RoboDK station: DensoAssembly.rdk

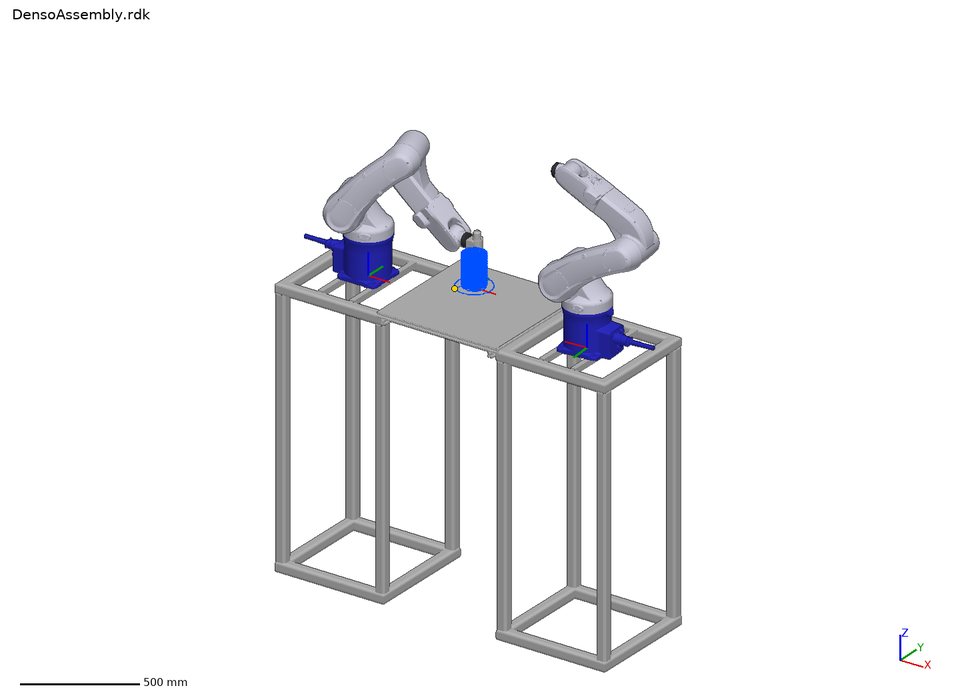
[picture v0: the station drawn from its stored meshes, robots at their saved joint values, targets as dots, program paths as lines]
Station DensoAssembly (saved by RoboDK 5.5.4). Poses are relative to the parent item; angles as X-Y-Z fixed-axis rotations.
Station parameters (name, value as stored): TAGS, ['Additive Manufacturing', 'Additive manufacturing']
  - frame Denso VS-6577G-B Base at (0, -10, -20) mm
    - robot Denso VS-6577G-B: 6 axes, payload 7 kg, reach 854 mm, repeatability 0.03 mm, weight 36 kg
        modified DH rows (alpha deg, a mm, theta deg, d mm): 0, 0, 0, 335; -90, 75, -90, 0; 0, 365, -90, 0; -90, 90, 0, 405; 90, 0, 0, 0; -90, 0, 0, 80
        joint limits [-170, -100, -119, -190, -120, -360] to [170, 135, 169, 190, 120, 360]; home [0, 0, 90, 0, 0, 0]; saved at [-161.491, -43.825, -94.782, 24.049, 51.169, -15.633]
      - tool NCRDK, TCP at (55, 0, 30) mm, rotated rx 0 ry 90 rz 0 deg, size 57.1 x 107.2 x 69.8 mm, geometry from NCRDK.STL
    - object Table 1400x800x800mm at (-100, 160, 0) mm, size 1420 x 820 x 800 mm, geometry from Table-1400x800x800mm.sld
    - object RobotStand_SWP at (50, -240, -710) mm, size 609.6 x 1373.2 x 1689.1 mm, geometry from RobotStand_SWP.STEP
  - frame Reference at (454.66, 114.92, 0) mm
    - object Part at (0, 0, 0) mm, size 120 x 120 x 160 mm, geometry from part.sld
  - machining project Print3D settings: C:/Users/Albert/AppData/Local/Temp/Part.stl | rotZ(0) | rotX(0)*rotY(0) | rotZ(0)
  - program Print3D (7572 instructions, listed below)
  - Python program Extruder (listed below)
  - Python program SimulateFinalResult (listed below)
  - frame Denso VS-6577G-B Base at (1145.1, -47.51, -20) mm, rotated rx 0 ry 0 rz -175.68 deg
    - robot Denso VS-6577G-B: 6 axes, payload 7 kg, reach 854 mm, repeatability 0.03 mm, weight 36 kg
        modified DH rows (alpha deg, a mm, theta deg, d mm): 0, 0, 0, 335; -90, 75, -90, 0; 0, 365, -90, 0; -90, 90, 0, 405; 90, 0, 0, 0; -90, 0, 0, 80
        joint limits [-170, -100, -119, -190, -120, -360] to [170, 135, 169, 190, 120, 360]; home [0, 0, 90, 0, 0, 0]; saved at [0, -58.32, 121.453, 0, 26.867, 0]
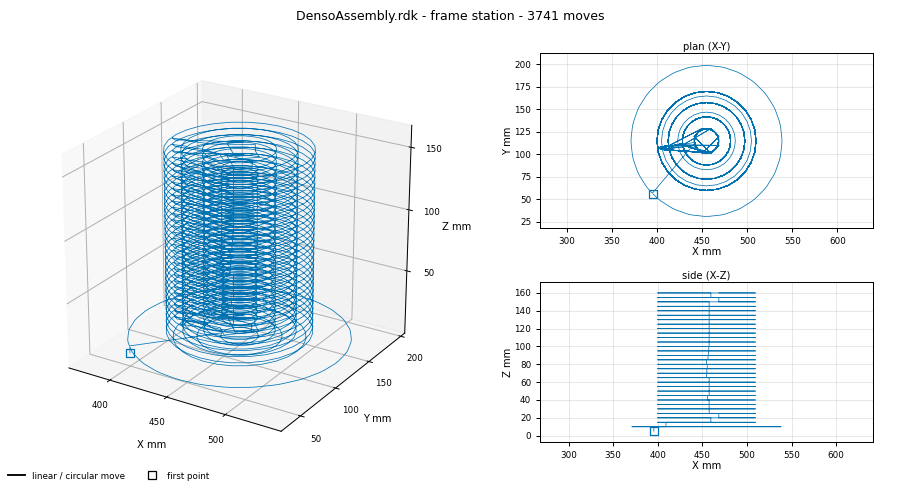
[picture p0: tool path of DensoAssembly.rdk in frame station, 3741 of 3741 moves have a stored position in this frame; points joined in program order, loops and branches not executed]

--- program Print3D (robot Denso VS-6577G-B) ---
  Set speed (83.3 mm/s)
  Set speed (1000.0 mm/s)
  Set Ref.: Reference
  Set Tool: NCRDK
  Show NCRDK
  MoveJ 1 to (-59.03, -59.03, 5) mm, rotated rx 180 ry 0 rz 180 deg; joints [-167.009, -64.344, -97.717, 13.631, 72.535, -4.163]
  MoveL 2 to (-59.03, -59.03, 5) mm, rotated rx 180 ry 0 rz 180 deg; joints [-167.009, -64.344, -97.717, 13.631, 72.535, -4.163]
  Call Extruder(-1)
  MoveL 3 to (-59.03, -59.03, 5) mm, rotated rx 180 ry 0 rz 180 deg; joints [-167.009, -64.344, -97.717, 13.631, 72.535, -4.163]
  Call Extruder(0.00000)
  Set speed (130.0 mm/s)
  MoveL 4 to (-59.03, -59.03, 10) mm, rotated rx 180 ry 0 rz 180 deg; joints [-167.009, -63.51, -98.227, 13.655, 72.22, -4.243]
  Call Extruder(-2.00000)
  Set speed (40.0 mm/s)
  MoveL 5 to (-59.03, -59.03, 10) mm, rotated rx 180 ry 0 rz 180 deg; joints [-167.009, -63.51, -98.227, 13.655, 72.22, -4.243]
  Call Extruder(0.00000)
  Set speed (130.0 mm/s)
  MoveL 6 to (-59.03, -59.03, 10) mm, rotated rx 180 ry 0 rz 180 deg; joints [-167.009, -63.51, -98.227, 13.655, 72.22, -4.243]
  Call Extruder(2.00000)
  Set speed (40.0 mm/s)
  MoveL 7 to (-59.03, -59.03, 10) mm, rotated rx 180 ry 0 rz 180 deg; joints [-167.009, -63.51, -98.227, 13.655, 72.22, -4.243]
  Call Extruder(25.86117)
  Set speed (30.0 mm/s)
  MoveL 8 to (-54.28, -63.78, 10) mm, rotated rx 180 ry 0 rz 180 deg; joints [-168.109, -63.573, -97.687, 12.537, 71.677, -3.999]
  Call Extruder(44.83322)
  MoveL 9 to (-50.1, -67.11, 10) mm, rotated rx 180 ry 0 rz 180 deg; joints [-168.895, -63.638, -97.171, 11.741, 71.182, -3.835]
  Call Extruder(92.55677)
  MoveL 10 to (-38.72, -74.26, 10) mm, rotated rx 180 ry 0 rz 176 deg; joints [-169.213, -63.884, -95.415, 15.759, 70.015, -5.509]
  Call Extruder(111.53101)
  MoveL 11 to (-33.91, -76.57, 10) mm, rotated rx 180 ry 0 rz 176 deg; joints [-169.789, -63.989, -94.75, 15.203, 69.419, -5.457]
  Call Extruder(159.25391)
  MoveL 12 to (-21.23, -81.01, 10) mm, rotated rx 180 ry 0 rz 172 deg; joints [-169.657, -64.367, -92.58, 19.815, 68.18, -7.628]
  Call Extruder(178.22553)
  MoveL 13 to (-16.02, -82.2, 10) mm, rotated rx 180 ry 0 rz 168 deg; joints [-168.792, -64.603, -91.363, 25.148, 68.018, -9.967]
  Call Extruder(225.94862)
  MoveL 14 to (-2.67, -83.7, 10) mm, rotated rx -180 ry 0 rz 168 deg; joints [-169.458, -65.044, -89.278, 24.729, 66.409, -10.444]
  Call Extruder(244.92246)
  MoveL 15 to (2.67, -83.7, 10) mm, rotated rx 180 ry 0 rz 168 deg; joints [-169.615, -65.24, -88.41, 24.684, 65.77, -10.682]
  Call Extruder(246.41380)
  MoveL 16 to (3.09, -83.66, 10) mm, rotated rx 180 ry 0 rz 168 deg; joints [-169.62, -65.256, -88.341, 24.689, 65.72, -10.704]
  Call Extruder(292.64546)
  MoveL 17 to (16.02, -82.2, 10) mm, rotated rx 180 ry 0 rz 168 deg; joints [-169.759, -65.781, -86.16, 24.862, 64.19, -11.406]
  Call Extruder(311.61718)
  MoveL 18 to (21.23, -81.01, 10) mm, rotated rx 180 ry 0 rz 168 deg; joints [-169.722, -66.013, -85.248, 25.044, 63.581, -11.744]
  Call Extruder(359.33987)
  MoveL 19 to (33.91, -76.57, 10) mm, rotated rx -180 ry 0 rz 168 deg; joints [-169.411, -66.628, -82.943, 25.757, 62.12, -12.714]
  Call Extruder(378.31438)
  MoveL 20 to (38.72, -74.26, 10) mm, rotated rx -180 ry 0 rz 168 deg; joints [-169.208, -66.882, -82.031, 26.136, 61.575, -13.147]
  Call Extruder(426.03771)
  MoveL 21 to (50.1, -67.11, 10) mm, rotated rx -180 ry 0 rz 172 deg; joints [-169.533, -67.389, -80.276, 21.566, 59.513, -11.339]
  Call Extruder(445.00995)
  MoveL 22 to (54.28, -63.78, 10) mm, rotated rx 180 ry 0 rz 172 deg; joints [-169.179, -67.643, -79.418, 22.103, 59.025, -11.806]
  Call Extruder(492.73236)
  MoveL 23 to (63.78, -54.28, 10) mm, rotated rx 180 ry 0 rz 176 deg; joints [-169.152, -68.143, -77.78, 17.748, 57.208, -9.834]
  Call Extruder(511.70474)
  MoveL 24 to (67.11, -50.1, 10) mm, rotated rx -180 ry 0 rz -180 deg; joints [-169.701, -68.281, -77.339, 12.417, 56.249, -6.974]
  Call Extruder(559.42802)
  MoveL 25 to (74.26, -38.72, 10) mm, rotated rx 180 ry 0 rz 180 deg; joints [-168.372, -68.831, -75.608, 14.195, 55.276, -8.199]
  Call Extruder(578.40244)
  MoveL 26 to (76.57, -33.91, 10) mm, rotated rx 180 ry 0 rz 180 deg; joints [-167.808, -69.033, -74.985, 14.95, 54.951, -8.718]
  Call Extruder(626.12508)
  MoveL 27 to (81.01, -21.23, 10) mm, rotated rx 180 ry 0 rz 180 deg; joints [-166.309, -69.49, -73.602, 16.944, 54.305, -10.08]
  Call Extruder(645.09694)
  MoveL 28 to (82.2, -16.02, 10) mm, rotated rx 180 ry 0 rz -180 deg; joints [-165.688, -69.648, -73.131, 17.765, 54.118, -10.635]
  Call Extruder(692.81987)
  MoveL 29 to (83.7, -2.67, 10) mm, rotated rx -180 ry 0 rz -180 deg; joints [-164.071, -69.976, -72.16, 19.875, 53.828, -12.044]
  Call Extruder(711.79372)
  MoveL 30 to (83.7, 2.67, 10) mm, rotated rx 180 ry 0 rz 180 deg; joints [-163.413, -70.078, -71.864, 20.722, 53.786, -12.599]
  Call Extruder(759.51663)
  MoveL 31 to (82.2, 16.02, 10) mm, rotated rx 180 ry 0 rz 180 deg; joints [-161.727, -70.253, -71.354, 22.845, 53.862, -13.953]
  Call Extruder(778.48846)
  MoveL 32 to (81.01, 21.23, 10) mm, rotated rx -180 ry 0 rz -180 deg; joints [-161.05, -70.29, -71.247, 23.678, 53.964, -14.465]
  Call Extruder(826.21114)
  MoveL 33 to (76.57, 33.91, 10) mm, rotated rx 180 ry 0 rz 180 deg; joints [-159.34, -70.299, -71.222, 25.719, 54.394, -15.666]
  Call Extruder(845.18561)
  MoveL 34 to (74.26, 38.72, 10) mm, rotated rx -180 ry 0 rz 180 deg; joints [-158.662, -70.268, -71.31, 26.502, 54.631, -16.099]
  Call Extruder(892.90887)
  MoveL 35 to (67.11, 50.1, 10) mm, rotated rx 180 ry 0 rz 180 deg; joints [-156.971, -70.109, -71.773, 28.382, 55.383, -17.063]
  Call Extruder(911.88119)
  MoveL 36 to (63.78, 54.28, 10) mm, rotated rx 180 ry 0 rz 180 deg; joints [-156.31, -70.014, -72.051, 29.087, 55.739, -17.389]
  Call Extruder(959.60361)
  MoveL 37 to (54.28, 63.78, 10) mm, rotated rx 180 ry 0 rz 180 deg; joints [-154.685, -69.699, -72.978, 30.745, 56.764, -18.056]
  Call Extruder(978.57593)
  MoveL 38 to (50.1, 67.11, 10) mm, rotated rx 180 ry 0 rz -180 deg; joints [-154.059, -69.547, -73.432, 31.353, 57.218, -18.257]
  Call Extruder(1026.29918)
  MoveL 39 to (38.72, 74.26, 10) mm, rotated rx -180 ry 0 rz 180 deg; joints [-152.546, -69.101, -74.778, 32.748, 58.459, -18.595]
  Call Extruder(1045.27367)
  MoveL 40 to (33.91, 76.57, 10) mm, rotated rx -180 ry 0 rz 180 deg; joints [-151.975, -68.903, -75.386, 33.246, 58.986, -18.663]
  Call Extruder(1092.99635)
  MoveL 41 to (21.23, 81.01, 10) mm, rotated rx -180 ry 0 rz -180 deg; joints [-150.627, -68.36, -77.086, 34.348, 60.378, -18.664]
  Call Extruder(1111.96805)
  MoveL 42 to (16.02, 82.2, 10) mm, rotated rx 180 ry 0 rz 180 deg; joints [-150.133, -68.131, -77.821, 34.725, 60.953, -18.599]
  Call Extruder(1159.69109)
  MoveL 43 to (2.67, 83.7, 10) mm, rotated rx 180 ry 0 rz -180 deg; joints [-149.008, -67.53, -79.796, 35.511, 62.434, -18.275]
  Call Extruder(1178.66494)
  MoveL 44 to (-2.67, 83.7, 10) mm, rotated rx 180 ry 0 rz 180 deg; joints [-148.615, -67.286, -80.624, 35.756, 63.03, -18.085]
  Call Extruder(1226.38787)
  MoveL 45 to (-16.02, 82.2, 10) mm, rotated rx 180 ry 0 rz -180 deg; joints [-147.779, -66.671, -82.786, 36.196, 64.538, -17.464]
  Call Extruder(1245.35974)
  MoveL 46 to (-21.23, 81.01, 10) mm, rotated rx -180 ry 0 rz -180 deg; joints [-147.514, -66.43, -83.669, 36.297, 65.134, -17.164]
  Call Extruder(1293.08238)
  MoveL 47 to (-33.91, 76.57, 10) mm, rotated rx 180 ry 0 rz 180 deg; joints [-147.039, -65.841, -85.922, 36.354, 66.611, -16.287]
  Call Extruder(1312.05679)
  MoveL 48 to (-38.72, 74.26, 10) mm, rotated rx -180 ry 0 rz 180 deg; joints [-146.933, -65.618, -86.82, 36.294, 67.184, -15.896]
  Call Extruder(1359.78007)
  MoveL 49 to (-50.1, 67.11, 10) mm, rotated rx -180 ry 0 rz 180 deg; joints [-146.898, -65.092, -89.06, 35.92, 68.579, -14.819]
  Call Extruder(1378.75242)
  MoveL 50 to (-54.28, 63.78, 10) mm, rotated rx 180 ry 0 rz -180 deg; joints [-146.982, -64.901, -89.932, 35.678, 69.11, -14.361]
  Call Extruder(1380.24377)
  MoveL 51 to (-54.57, 63.48, 10) mm, rotated rx 180 ry 0 rz 180 deg; joints [-146.997, -64.886, -89.999, 35.652, 69.149, -14.322]
  Call Extruder(1426.47485)
  MoveL 52 to (-63.78, 54.28, 10) mm, rotated rx 180 ry 0 rz -180 deg; joints [-147.462, -64.468, -92.052, 34.822, 70.373, -13.151]
  Call Extruder(1445.44710)
  MoveL 53 to (-67.11, 50.1, 10) mm, rotated rx 180 ry 0 rz -180 deg; joints [-147.764, -64.316, -92.854, 34.38, 70.841, -12.656]
  Call Extruder(1493.17037)
  MoveL 54 to (-74.26, 38.72, 10) mm, rotated rx 180 ry 0 rz 180 deg; joints [-148.817, -63.99, -94.742, 33.001, 71.922, -11.394]
  Call Extruder(1512.14494)
  MoveL 55 to (-76.57, 33.91, 10) mm, rotated rx 180 ry 0 rz 180 deg; joints [-149.354, -63.882, -95.431, 32.347, 72.307, -10.895]
  Call Extruder(1559.86760)
  MoveL 56 to (-81.01, 21.23, 10) mm, rotated rx -180 ry 0 rz -180 deg; joints [-150.998, -63.662, -96.979, 30.438, 73.148, -9.667]
  Call Extruder(1578.83925)
  MoveL 57 to (-82.2, 16.02, 10) mm, rotated rx 180 ry 0 rz -180 deg; joints [-151.763, -63.595, -97.512, 29.58, 73.425, -9.198]
  Call Extruder(1626.56228)
  MoveL 58 to (-83.7, 2.67, 10) mm, rotated rx -180 ry 0 rz 180 deg; joints [-153.943, -63.467, -98.621, 27.197, 73.961, -8.081]
  Call Extruder(1645.53608)
  MoveL 59 to (-83.7, -2.67, 10) mm, rotated rx -180 ry 0 rz -180 deg; joints [-154.897, -63.432, -98.963, 26.175, 74.104, -7.667]
  Call Extruder(1693.25913)
  MoveL 60 to (-82.2, -16.02, 10) mm, rotated rx -180 ry 0 rz 180 deg; joints [-157.465, -63.375, -99.554, 23.464, 74.267, -6.713]
  Call Extruder(1712.23091)
  MoveL 61 to (-81.01, -21.23, 10) mm, rotated rx -180 ry 0 rz 180 deg; joints [-158.53, -63.363, -99.678, 22.352, 74.25, -6.368]
  Call Extruder(1759.95353)
  MoveL 62 to (-76.57, -33.91, 10) mm, rotated rx 180 ry 0 rz 180 deg; joints [-161.248, -63.361, -99.707, 19.539, 73.991, -5.59]
  Call Extruder(1778.92790)
  MoveL 63 to (-74.26, -38.72, 10) mm, rotated rx 180 ry 0 rz 180 deg; joints [-162.318, -63.37, -99.605, 18.438, 73.802, -5.314]
  Call Extruder(1826.65135)
  MoveL 64 to (-67.11, -50.1, 10) mm, rotated rx 180 ry 0 rz 180 deg; joints [-164.913, -63.421, -99.068, 15.785, 73.111, -4.695]
  Call Extruder(1845.62336)
  MoveL 65 to (-63.78, -54.28, 10) mm, rotated rx 180 ry 0 rz -180 deg; joints [-165.882, -63.454, -98.747, 14.798, 72.756, -4.478]
  Call Extruder(1864.15697)
  MoveL 66 to (-60.09, -57.97, 10) mm, rotated rx -180 ry 0 rz 180 deg; joints [-166.759, -63.497, -98.345, 13.908, 72.341, -4.296]
  Call Extruder(1862.15697)
  Set speed (40.0 mm/s)
  MoveL 67 to (-60.09, -57.97, 10) mm, rotated rx -180 ry 0 rz 180 deg; joints [-166.759, -63.497, -98.345, 13.908, 72.341, -4.296]
  Call Extruder(0.00000)
  Set speed (130.0 mm/s)
  MoveL 68 to (-13.65, -3.12, 10) mm, rotated rx -180 ry 0 rz 180 deg; joints [-159.797, -65.133, -88.882, 22.263, 65.721, -9.555]
  Call Extruder(2.00000)
  Set speed (40.0 mm/s)
  MoveL 69 to (-13.65, -3.12, 10) mm, rotated rx -180 ry 0 rz 180 deg; joints [-159.797, -65.133, -88.882, 22.263, 65.721, -9.555]
  Call Extruder(13.13706)
  Set speed (30.0 mm/s)
  MoveL 70 to (-12.62, -6.08, 10) mm, rotated rx 180 ry 0 rz 180 deg; joints [-160.306, -65.131, -88.888, 21.711, 65.641, -9.326]
  Call Extruder(24.27428)
  MoveL 71 to (-10.95, -8.73, 10) mm, rotated rx -180 ry 0 rz 180 deg; joints [-160.802, -65.157, -88.774, 21.188, 65.48, -9.139]
  Call Extruder(35.41276)
  MoveL 72 to (-8.73, -10.95, 10) mm, rotated rx -180 ry 0 rz 180 deg; joints [-161.258, -65.209, -88.546, 20.721, 65.244, -9.002]
  Call Extruder(46.54998)
  MoveL 73 to (-6.08, -12.62, 10) mm, rotated rx 180 ry 0 rz -180 deg; joints [-161.649, -65.285, -88.217, 20.337, 64.945, -8.92]
  Call Extruder(57.68705)
  MoveL 74 to (-3.12, -13.65, 10) mm, rotated rx -180 ry 0 rz 180 deg; joints [-161.955, -65.382, -87.802, 20.055, 64.6, -8.899]
  Call Extruder(68.82500)
  MoveL 75 to (0, -14, 10) mm, rotated rx -180 ry 0 rz 180 deg; joints [-162.16, -65.496, -87.324, 19.889, 64.225, -8.94]
  Call Extruder(79.96296)
  MoveL 76 to (3.12, -13.65, 10) mm, rotated rx -180 ry 0 rz 180 deg; joints [-162.258, -65.621, -86.806, 19.847, 63.842, -9.042]
  Call Extruder(91.10003)
  MoveL 77 to (6.08, -12.62, 10) mm, rotated rx 180 ry 0 rz 180 deg; joints [-162.244, -65.752, -86.276, 19.929, 63.468, -9.2]
  Call Extruder(102.23724)
  MoveL 78 to (8.73, -10.95, 10) mm, rotated rx 180 ry 0 rz -180 deg; joints [-162.124, -65.882, -85.759, 20.128, 63.124, -9.408]
  Call Extruder(113.37572)
  MoveL 79 to (10.95, -8.73, 10) mm, rotated rx 180 ry 0 rz 180 deg; joints [-161.905, -66.004, -85.281, 20.434, 62.826, -9.656]
  Call Extruder(124.51294)
  MoveL 80 to (12.62, -6.08, 10) mm, rotated rx -180 ry 0 rz 180 deg; joints [-161.6, -66.112, -84.866, 20.828, 62.59, -9.933]
  Call Extruder(135.65003)
  MoveL 81 to (13.65, -3.12, 10) mm, rotated rx 180 ry 0 rz 180 deg; joints [-161.224, -66.199, -84.533, 21.291, 62.427, -10.225]
  Call Extruder(146.78796)
  MoveL 82 to (14, 0, 10) mm, rotated rx 180 ry 0 rz 180 deg; joints [-160.796, -66.261, -84.3, 21.799, 62.345, -10.516]
  Call Extruder(157.92590)
  MoveL 83 to (13.65, 3.12, 10) mm, rotated rx 180 ry 0 rz 180 deg; joints [-160.336, -66.293, -84.178, 22.328, 62.347, -10.792]
  Call Extruder(169.06301)
  MoveL 84 to (12.62, 6.08, 10) mm, rotated rx 180 ry 0 rz 180 deg; joints [-159.864, -66.295, -84.172, 22.852, 62.432, -11.036]
  Call Extruder(180.20021)
  MoveL 85 to (10.95, 8.73, 10) mm, rotated rx 180 ry 0 rz 180 deg; joints [-159.401, -66.265, -84.283, 23.346, 62.597, -11.236]
  Call Extruder(191.33869)
  MoveL 86 to (8.73, 10.95, 10) mm, rotated rx -180 ry 0 rz -180 deg; joints [-158.969, -66.206, -84.506, 23.79, 62.831, -11.381]
  Call Extruder(202.47589)
  MoveL 87 to (6.08, 12.62, 10) mm, rotated rx 180 ry 0 rz -180 deg; joints [-158.587, -66.122, -84.829, 24.16, 63.124, -11.463]
  Call Extruder(213.61299)
  MoveL 88 to (3.12, 13.65, 10) mm, rotated rx 180 ry 0 rz 180 deg; joints [-158.274, -66.016, -85.237, 24.441, 63.462, -11.478]
  Call Extruder(224.75094)
  MoveL 89 to (0, 14, 10) mm, rotated rx 180 ry 0 rz -180 deg; joints [-158.046, -65.895, -85.709, 24.618, 63.827, -11.426]
  Call Extruder(235.88887)
  MoveL 90 to (-3.12, 13.65, 10) mm, rotated rx 180 ry 0 rz 180 deg; joints [-157.916, -65.765, -86.224, 24.682, 64.203, -11.31]
  Call Extruder(247.02595)
  MoveL 91 to (-6.08, 12.62, 10) mm, rotated rx 180 ry 0 rz -180 deg; joints [-157.892, -65.634, -86.754, 24.629, 64.57, -11.137]
  Call Extruder(258.16319)
  MoveL 92 to (-8.73, 10.95, 10) mm, rotated rx -180 ry 0 rz 180 deg; joints [-157.978, -65.508, -87.274, 24.458, 64.912, -10.916]
  Call Extruder(269.30166)
  MoveL 93 to (-10.95, 8.73, 10) mm, rotated rx -180 ry 0 rz 180 deg; joints [-158.173, -65.392, -87.757, 24.176, 65.211, -10.66]
  Call Extruder(280.43886)
  MoveL 94 to (-12.62, 6.08, 10) mm, rotated rx 180 ry 0 rz 180 deg; joints [-158.469, -65.294, -88.179, 23.795, 65.452, -10.381]
  Call Extruder(291.57594)
  MoveL 95 to (-13.65, 3.12, 10) mm, rotated rx 180 ry 0 rz 180 deg; joints [-158.852, -65.215, -88.518, 23.334, 65.623, -10.095]
  Call Extruder(302.71390)
  MoveL 96 to (-14, 0, 10) mm, rotated rx 180 ry 0 rz 180 deg; joints [-159.303, -65.161, -88.756, 22.814, 65.714, -9.816]
  Call Extruder(308.52395)
  MoveL 97 to (-13.82, -1.63, 10) mm, rotated rx 180 ry 0 rz 180 deg; joints [-159.56, -65.146, -88.822, 22.527, 65.718, -9.68]
  Set speed (130.0 mm/s)
  MoveL 98 to (-31.39, -5.11, 10) mm, rotated rx -180 ry 0 rz 180 deg; joints [-159.07, -64.537, -91.697, 22.68, 67.888, -8.939]
  Call Extruder(315.66877)
  Set speed (30.0 mm/s)
  MoveL 99 to (-31.17, -7.11, 10) mm, rotated rx -180 ry 0 rz 180 deg; joints [-159.404, -64.521, -91.777, 22.314, 67.896, -8.779]
  Call Extruder(341.09651)
  MoveL 100 to (-28.8, -13.87, 10) mm, rotated rx 180 ry 0 rz 180 deg; joints [-160.628, -64.518, -91.791, 21.005, 67.725, -8.281]
  Call Extruder(366.52461)
  MoveL 101 to (-24.99, -19.93, 10) mm, rotated rx 180 ry 0 rz 180 deg; joints [-161.818, -64.571, -91.526, 19.761, 67.358, -7.874]
  Call Extruder(391.95312)
  MoveL 102 to (-19.93, -25, 10) mm, rotated rx -180 ry 0 rz -180 deg; joints [-162.895, -64.677, -90.996, 18.661, 66.814, -7.574]
  Call Extruder(417.38123)
  MoveL 103 to (-13.87, -28.8, 10) mm, rotated rx 180 ry 0 rz -180 deg; joints [-163.797, -64.837, -90.232, 17.768, 66.122, -7.391]
  Call Extruder(442.80898)
  MoveL 104 to (-7.11, -31.17, 10) mm, rotated rx -180 ry 0 rz -180 deg; joints [-164.477, -65.045, -89.275, 17.13, 65.32, -7.333]
  Call Extruder(468.23739)
  MoveL 105 to (0, -31.97, 10) mm, rotated rx 180 ry 0 rz 180 deg; joints [-164.906, -65.295, -88.175, 16.775, 64.452, -7.407]
  Call Extruder(493.66579)
  MoveL 106 to (7.11, -31.17, 10) mm, rotated rx -180 ry 0 rz 180 deg; joints [-165.076, -65.576, -86.99, 16.715, 63.565, -7.614]
  Call Extruder(519.09356)
  MoveL 107 to (13.87, -28.8, 10) mm, rotated rx 180 ry 0 rz 180 deg; joints [-164.992, -65.877, -85.78, 16.941, 62.706, -7.952]
  Call Extruder(544.52164)
  MoveL 108 to (19.93, -24.99, 10) mm, rotated rx 180 ry 0 rz -180 deg; joints [-164.672, -66.18, -84.604, 17.434, 61.918, -8.409]
  Call Extruder(569.95016)
  MoveL 109 to (25, -19.93, 10) mm, rotated rx 180 ry 0 rz 180 deg; joints [-164.144, -66.47, -83.521, 18.159, 61.242, -8.968]
  Call Extruder(595.37826)
  MoveL 110 to (28.8, -13.87, 10) mm, rotated rx -180 ry 0 rz 180 deg; joints [-163.439, -66.728, -82.581, 19.075, 60.71, -9.602]
  Call Extruder(620.80602)
  MoveL 111 to (31.17, -7.11, 10) mm, rotated rx -180 ry 0 rz -180 deg; joints [-162.595, -66.939, -81.831, 20.133, 60.348, -10.28]
  Call Extruder(646.23442)
  MoveL 112 to (31.97, 0, 10) mm, rotated rx 180 ry 0 rz -180 deg; joints [-161.65, -67.089, -81.305, 21.279, 60.17, -10.964]
  Call Extruder(671.66281)
  MoveL 113 to (31.17, 7.11, 10) mm, rotated rx 180 ry 0 rz 180 deg; joints [-160.642, -67.169, -81.029, 22.46, 60.185, -11.615]
  Call Extruder(697.09060)
  MoveL 114 to (28.8, 13.87, 10) mm, rotated rx 180 ry 0 rz 180 deg; joints [-159.613, -67.172, -81.016, 23.622, 60.389, -12.194]
  Call Extruder(722.51868)
  MoveL 115 to (25, 19.93, 10) mm, rotated rx 180 ry 0 rz 180 deg; joints [-158.601, -67.1, -81.266, 24.715, 60.769, -12.667]
  Call Extruder(747.94720)
  MoveL 116 to (19.93, 24.99, 10) mm, rotated rx -180 ry 0 rz 180 deg; joints [-157.648, -66.957, -81.768, 25.693, 61.306, -13.007]
  Call Extruder(773.37528)
  MoveL 117 to (13.87, 28.8, 10) mm, rotated rx -180 ry 0 rz 180 deg; joints [-156.791, -66.751, -82.498, 26.516, 61.97, -13.195]
  Call Extruder(798.80307)
  MoveL 118 to (7.11, 31.17, 10) mm, rotated rx -180 ry 0 rz 180 deg; joints [-156.072, -66.497, -83.42, 27.149, 62.731, -13.222]
  Call Extruder(824.23147)
  MoveL 119 to (0, 31.97, 10) mm, rotated rx 180 ry 0 rz -180 deg; joints [-155.524, -66.21, -84.492, 27.564, 63.552, -13.088]
  Call Extruder(849.65986)
  MoveL 120 to (-7.11, 31.17, 10) mm, rotated rx -180 ry 0 rz 180 deg; joints [-155.182, -65.907, -85.661, 27.738, 64.396, -12.803]
  Call Extruder(875.08762)
  MoveL 121 to (-13.87, 28.8, 10) mm, rotated rx -180 ry 0 rz 180 deg; joints [-155.074, -65.606, -86.87, 27.657, 65.223, -12.387]
  Call Extruder(900.51573)
  MoveL 122 to (-19.93, 25, 10) mm, rotated rx 180 ry 0 rz 180 deg; joints [-155.218, -65.321, -88.06, 27.313, 65.997, -11.864]
  Call Extruder(925.94424)
  MoveL 123 to (-25, 19.93, 10) mm, rotated rx 180 ry 0 rz 180 deg; joints [-155.622, -65.068, -89.171, 26.71, 66.68, -11.265]
  Call Extruder(951.37232)
  MoveL 124 to (-28.8, 13.87, 10) mm, rotated rx -180 ry 0 rz -180 deg; joints [-156.278, -64.855, -90.145, 25.867, 67.238, -10.625]
  Call Extruder(976.80009)
  MoveL 125 to (-31.17, 7.11, 10) mm, rotated rx -180 ry 0 rz 180 deg; joints [-157.16, -64.691, -90.93, 24.817, 67.642, -9.977]
  Call Extruder(1002.22850)
  MoveL 126 to (-31.97, 0, 10) mm, rotated rx 180 ry 0 rz 180 deg; joints [-158.222, -64.579, -91.485, 23.611, 67.866, -9.352]
  Call Extruder(1015.18419)
  MoveL 127 to (-31.56, -3.63, 10) mm, rotated rx -180 ry 0 rz -180 deg; joints [-158.823, -64.549, -91.637, 22.951, 67.882, -9.059]
  Set speed (130.0 mm/s)
  MoveL 128 to (-49.14, -7.11, 10) mm, rotated rx -180 ry 0 rz 180 deg; joints [-158.265, -64.042, -94.421, 23.199, 70.062, -8.315]
  Call Extruder(1029.47382)
  Set speed (30.0 mm/s)
  MoveL 129 to (-48.69, -11.11, 10) mm, rotated rx -180 ry 0 rz 180 deg; joints [-158.966, -64.016, -94.582, 22.442, 70.087, -8.007]
  Call Extruder(1069.19224)
  MoveL 130 to (-44.99, -21.67, 10) mm, rotated rx -180 ry 0 rz 180 deg; joints [-160.987, -64.012, -94.604, 20.307, 69.835, -7.27]
  Call Extruder(1108.91123)
  MoveL 131 to (-39.04, -31.13, 10) mm, rotated rx 180 ry 0 rz -180 deg; joints [-162.939, -64.083, -94.18, 18.283, 69.265, -6.672]
  Call Extruder(1148.62978)
  MoveL 132 to (-31.13, -39.04, 10) mm, rotated rx 180 ry 0 rz 180 deg; joints [-164.681, -64.229, -93.336, 16.508, 68.403, -6.225]
  Call Extruder(1188.34877)
  MoveL 133 to (-21.67, -44.99, 10) mm, rotated rx -180 ry 0 rz 180 deg; joints [-166.1, -64.454, -92.122, 15.094, 67.301, -5.942]
  Call Extruder(1228.06720)
  MoveL 134 to (-11.11, -48.68, 10) mm, rotated rx 180 ry 0 rz 180 deg; joints [-167.125, -64.757, -90.609, 14.115, 66.025, -5.834]
  Call Extruder(1267.78606)
  MoveL 135 to (0, -49.94, 10) mm, rotated rx 180 ry 0 rz 180 deg; joints [-167.725, -65.133, -88.88, 13.606, 64.649, -5.917]
  Call Extruder(1307.50491)
  MoveL 136 to (11.11, -48.69, 10) mm, rotated rx -180 ry 0 rz 180 deg; joints [-167.905, -65.568, -87.025, 13.571, 63.25, -6.201]
  Call Extruder(1347.22336)
  MoveL 137 to (21.67, -44.99, 10) mm, rotated rx 180 ry 0 rz 180 deg; joints [-167.691, -66.041, -85.137, 13.985, 61.901, -6.69]
  Call Extruder(1386.94233)
  MoveL 138 to (31.13, -39.04, 10) mm, rotated rx -180 ry 0 rz -180 deg; joints [-167.127, -66.527, -83.31, 14.806, 60.67, -7.377]
  Call Extruder(1426.66090)
  MoveL 139 to (39.04, -31.14, 10) mm, rotated rx -180 ry 0 rz 180 deg; joints [-166.264, -66.997, -81.628, 15.976, 59.619, -8.239]
  Call Extruder(1466.37987)
  MoveL 140 to (44.99, -21.67, 10) mm, rotated rx -180 ry 0 rz -180 deg; joints [-165.158, -67.419, -80.173, 17.427, 58.797, -9.236]
  Call Extruder(1506.09831)
  MoveL 141 to (48.69, -11.11, 10) mm, rotated rx -180 ry 0 rz 180 deg; joints [-163.862, -67.766, -79.01, 19.08, 58.243, -10.317]
  Call Extruder(1545.81716)
  MoveL 142 to (49.94, 0, 10) mm, rotated rx -180 ry 0 rz 180 deg; joints [-162.433, -68.015, -78.196, 20.853, 57.981, -11.419]
  Call Extruder(1585.53601)
  MoveL 143 to (48.69, 11.11, 10) mm, rotated rx -180 ry 0 rz 180 deg; joints [-160.922, -68.147, -77.769, 22.665, 58.019, -12.471]
  Call Extruder(1625.25448)
  MoveL 144 to (44.99, 21.67, 10) mm, rotated rx 180 ry 0 rz 180 deg; joints [-159.383, -68.153, -77.748, 24.433, 58.351, -13.408]
  Call Extruder(1664.97343)
  MoveL 145 to (39.04, 31.13, 10) mm, rotated rx 180 ry 0 rz 180 deg; joints [-157.867, -68.033, -78.136, 26.087, 58.955, -14.171]
  Call Extruder(1704.69201)
  MoveL 146 to (31.14, 39.04, 10) mm, rotated rx -180 ry 0 rz 180 deg; joints [-156.427, -67.796, -78.913, 27.564, 59.795, -14.714]
  Call Extruder(1744.41096)
  MoveL 147 to (21.67, 44.99, 10) mm, rotated rx -180 ry 0 rz 180 deg; joints [-155.116, -67.457, -80.043, 28.809, 60.829, -15.006]
  Call Extruder(1784.12943)
  MoveL 148 to (11.11, 48.69, 10) mm, rotated rx -180 ry 0 rz 180 deg; joints [-153.988, -67.041, -81.473, 29.78, 62.005, -15.035]
  Call Extruder(1823.84828)
  MoveL 149 to (0, 49.94, 10) mm, rotated rx 180 ry 0 rz -180 deg; joints [-153.099, -66.575, -83.135, 30.437, 63.269, -14.804]
  Call Extruder(1863.56714)
  MoveL 150 to (-11.11, 48.69, 10) mm, rotated rx 180 ry 0 rz 180 deg; joints [-152.503, -66.089, -84.952, 30.747, 64.565, -14.332]
  Call Extruder(1903.28558)
  MoveL 151 to (-21.67, 44.99, 10) mm, rotated rx -180 ry 0 rz 180 deg; joints [-152.252, -65.614, -86.837, 30.683, 65.838, -13.651]
  Call Extruder(1943.00455)
  MoveL 152 to (-31.13, 39.04, 10) mm, rotated rx 180 ry 0 rz -180 deg; joints [-152.391, -65.174, -88.7, 30.221, 67.032, -12.806]
  Call Extruder(1982.72311)
  MoveL 153 to (-39.04, 31.14, 10) mm, rotated rx -180 ry 0 rz 180 deg; joints [-152.949, -64.792, -90.446, 29.351, 68.097, -11.848]
  Call Extruder(2022.44207)
  MoveL 154 to (-44.99, 21.67, 10) mm, rotated rx 180 ry 0 rz 180 deg; joints [-153.933, -64.481, -91.984, 28.083, 68.98, -10.835]
  Call Extruder(2062.16053)
  MoveL 155 to (-48.68, 11.11, 10) mm, rotated rx 180 ry 0 rz -180 deg; joints [-155.315, -64.248, -93.231, 26.454, 69.633, -9.824]
  Call Extruder(2101.87939)
  MoveL 156 to (-49.94, 0, 10) mm, rotated rx 180 ry 0 rz 180 deg; joints [-157.029, -64.094, -94.115, 24.537, 70.014, -8.868]
  Call Extruder(2121.98071)
  MoveL 157 to (-49.3, -5.62, 10) mm, rotated rx 180 ry 0 rz 180 deg; joints [-158.005, -64.053, -94.359, 23.48, 70.052, -8.43]
  Set speed (130.0 mm/s)
  MoveL 158 to (-45.45, -8.72, 10) mm, rotated rx 180 ry 0 rz 180 deg; joints [-158.776, -64.117, -93.978, 22.713, 69.649, -8.282]
  MoveL 159 to (-45.45, -8.72, 15) mm, rotated rx -180 ry 0 rz 180 deg; joints [-158.776, -63.309, -94.467, 22.76, 69.354, -8.414]
  MoveL 160 to (-26.25, -4.54, 15) mm, rotated rx 180 ry 0 rz 180 deg; joints [-159.288, -63.909, -91.373, 22.599, 66.975, -9.247]
  Call Extruder(2124.21334)
  Set speed (60.0 mm/s)
  MoveL 161 to (-26.09, -5.96, 15) mm, rotated rx 180 ry 0 rz 180 deg; joints [-159.522, -63.897, -91.43, 22.341, 66.98, -9.13]
  Call Extruder(2133.57813)
  MoveL 162 to (-24.11, -11.61, 15) mm, rotated rx 180 ry 0 rz 180 deg; joints [-160.532, -63.895, -91.442, 21.255, 66.832, -8.701]
  Call Extruder(2142.94305)
  MoveL 163 to (-20.93, -16.69, 15) mm, rotated rx 180 ry 0 rz 180 deg; joints [-161.513, -63.941, -91.22, 20.225, 66.523, -8.35]
  Call Extruder(2152.30825)
  MoveL 164 to (-16.69, -20.93, 15) mm, rotated rx 180 ry 0 rz 180 deg; joints [-162.406, -64.036, -90.779, 19.311, 66.069, -8.09]
  Call Extruder(2161.67318)
  MoveL 165 to (-11.61, -24.12, 15) mm, rotated rx 180 ry 0 rz 180 deg; joints [-163.159, -64.177, -90.141, 18.566, 65.493, -7.931]
  Call Extruder(2171.03796)
  MoveL 166 to (-5.96, -26.09, 15) mm, rotated rx -180 ry 0 rz 180 deg; joints [-163.733, -64.358, -89.34, 18.029, 64.827, -7.882]
  Call Extruder(2180.40308)
  MoveL 167 to (0, -26.77, 15) mm, rotated rx 180 ry 0 rz 180 deg; joints [-164.103, -64.575, -88.42, 17.727, 64.106, -7.947]
  Call Extruder(2189.76818)
  MoveL 168 to (5.96, -26.09, 15) mm, rotated rx -180 ry 0 rz -180 deg; joints [-164.258, -64.817, -87.427, 17.668, 63.369, -8.126]
  Call Extruder(2199.13298)
  MoveL 169 to (11.61, -24.11, 15) mm, rotated rx 180 ry 0 rz 180 deg; joints [-164.201, -65.073, -86.412, 17.85, 62.655, -8.414]
  Call Extruder(2208.49789)
  MoveL 170 to (16.69, -20.93, 15) mm, rotated rx -180 ry 0 rz 180 deg; joints [-163.944, -65.33, -85.426, 18.255, 62, -8.803]
  Call Extruder(2217.86309)
  MoveL 171 to (20.93, -16.69, 15) mm, rotated rx -180 ry 0 rz -180 deg; joints [-163.508, -65.574, -84.516, 18.858, 61.437, -9.275]
  Call Extruder(2227.22802)
  MoveL 172 to (24.11, -11.61, 15) mm, rotated rx 180 ry 0 rz 180 deg; joints [-162.92, -65.791, -83.727, 19.624, 60.994, -9.809]
  Call Extruder(2236.59281)
  MoveL 173 to (26.09, -5.96, 15) mm, rotated rx -180 ry 0 rz -180 deg; joints [-162.209, -65.967, -83.096, 20.511, 60.692, -10.378]
  Call Extruder(2245.95792)
  MoveL 174 to (26.77, 0, 15) mm, rotated rx 180 ry 0 rz -180 deg; joints [-161.41, -66.092, -82.654, 21.476, 60.544, -10.95]
  Call Extruder(2255.32302)
  MoveL 175 to (26.09, 5.96, 15) mm, rotated rx 180 ry 0 rz 180 deg; joints [-160.556, -66.159, -82.422, 22.473, 60.557, -11.494]
  Call Extruder(2264.68782)
  MoveL 176 to (24.11, 11.61, 15) mm, rotated rx 180 ry 0 rz 180 deg; joints [-159.683, -66.162, -82.411, 23.456, 60.727, -11.978]
  Call Extruder(2274.05273)
  MoveL 177 to (20.93, 16.69, 15) mm, rotated rx -180 ry 0 rz 180 deg; joints [-158.826, -66.102, -82.622, 24.381, 61.045, -12.376]
  Call Extruder(2283.41794)
  MoveL 178 to (16.69, 20.93, 15) mm, rotated rx -180 ry 0 rz 180 deg; joints [-158.019, -65.982, -83.043, 25.209, 61.494, -12.663]
  Call Extruder(2292.78285)
  MoveL 179 to (11.61, 24.11, 15) mm, rotated rx -180 ry 0 rz 180 deg; joints [-157.299, -65.81, -83.657, 25.905, 62.051, -12.824]
  Call Extruder(2302.14766)
  MoveL 180 to (5.96, 26.09, 15) mm, rotated rx -180 ry 0 rz 180 deg; joints [-156.697, -65.597, -84.432, 26.437, 62.689, -12.851]
  Call Extruder(2311.51276)
  MoveL 181 to (0, 26.77, 15) mm, rotated rx -180 ry 0 rz 180 deg; joints [-156.245, -65.355, -85.331, 26.782, 63.377, -12.745]
  Call Extruder(2320.87786)
  MoveL 182 to (-5.96, 26.09, 15) mm, rotated rx 180 ry 0 rz -180 deg; joints [-155.969, -65.098, -86.313, 26.921, 64.084, -12.513]
  Call Extruder(2330.24266)
  MoveL 183 to (-11.61, 24.11, 15) mm, rotated rx 180 ry 0 rz 180 deg; joints [-155.891, -64.842, -87.327, 26.841, 64.776, -12.17]
  Call Extruder(2339.60758)
  MoveL 184 to (-16.69, 20.93, 15) mm, rotated rx -180 ry 0 rz -180 deg; joints [-156.025, -64.598, -88.324, 26.54, 65.422, -11.736]
  Call Extruder(2348.97278)
  MoveL 185 to (-20.93, 16.69, 15) mm, rotated rx -180 ry 0 rz 180 deg; joints [-156.374, -64.378, -89.254, 26.023, 65.989, -11.236]
  Call Extruder(2358.33769)
  MoveL 186 to (-24.11, 11.61, 15) mm, rotated rx -180 ry 0 rz 180 deg; joints [-156.928, -64.193, -90.068, 25.308, 66.45, -10.699]
  Call Extruder(2367.70249)
  MoveL 187 to (-26.09, 5.96, 15) mm, rotated rx -180 ry 0 rz -180 deg; joints [-157.665, -64.048, -90.724, 24.426, 66.781, -10.151]
  Call Extruder(2377.06760)
  MoveL 188 to (-26.77, 0, 15) mm, rotated rx -180 ry 0 rz -180 deg; joints [-158.546, -63.949, -91.186, 23.419, 66.961, -9.621]
  Call Extruder(2381.85633)
  MoveL 189 to (-26.42, -3.05, 15) mm, rotated rx -180 ry 0 rz 180 deg; joints [-159.044, -63.922, -91.313, 22.869, 66.971, -9.369]
  Set speed (130.0 mm/s)
  MoveL 190 to (-41.86, -6.3, 15) mm, rotated rx -180 ry 0 rz 180 deg; joints [-158.606, -63.428, -93.803, 23.02, 68.879, -8.705]
  Call Extruder(2386.85418)
  Set speed (60.0 mm/s)
  MoveL 191 to (-41.5, -9.47, 15) mm, rotated rx 180 ry 0 rz 180 deg; joints [-159.151, -63.405, -93.931, 22.426, 68.893, -8.453]
  Call Extruder(2401.74983)
  MoveL 192 to (-38.36, -18.47, 15) mm, rotated rx 180 ry 0 rz 180 deg; joints [-160.835, -63.401, -93.95, 20.636, 68.67, -7.8]
  Call Extruder(2416.64568)
  MoveL 193 to (-33.28, -26.54, 15) mm, rotated rx 180 ry 0 rz 180 deg; joints [-162.466, -63.468, -93.591, 18.937, 68.181, -7.267]
  Call Extruder(2431.54150)
  MoveL 194 to (-26.54, -33.28, 15) mm, rotated rx -180 ry 0 rz -180 deg; joints [-163.93, -63.604, -92.876, 17.441, 67.451, -6.87]
  Call Extruder(2446.43735)
  MoveL 195 to (-18.47, -38.36, 15) mm, rotated rx 180 ry 0 rz 180 deg; joints [-165.137, -63.81, -91.846, 16.24, 66.521, -6.62]
  Call Extruder(2461.33300)
  MoveL 196 to (-9.47, -41.5, 15) mm, rotated rx 180 ry 0 rz 180 deg; joints [-166.024, -64.084, -90.559, 15.398, 65.444, -6.529]
  Call Extruder(2476.22889)
  MoveL 197 to (0, -42.57, 15) mm, rotated rx 180 ry 0 rz 180 deg; joints [-166.562, -64.417, -89.086, 14.948, 64.283, -6.608]
  Call Extruder(2491.12475)
  MoveL 198 to (9.47, -41.5, 15) mm, rotated rx 180 ry 0 rz 180 deg; joints [-166.745, -64.798, -87.504, 14.898, 63.1, -6.864]
  Call Extruder(2506.02041)
  MoveL 199 to (18.47, -38.36, 15) mm, rotated rx 180 ry 0 rz 180 deg; joints [-166.591, -65.208, -85.891, 15.233, 61.958, -7.295]
  Call Extruder(2520.91626)
  MoveL 200 to (26.54, -33.29, 15) mm, rotated rx -180 ry 0 rz 180 deg; joints [-166.133, -65.625, -84.329, 15.918, 60.915, -7.893]
  Call Extruder(2535.81208)
  MoveL 201 to (33.29, -26.54, 15) mm, rotated rx 180 ry 0 rz 180 deg; joints [-165.409, -66.025, -82.89, 16.907, 60.023, -8.635]
  Call Extruder(2550.70793)
  MoveL 202 to (38.36, -18.47, 15) mm, rotated rx 180 ry 0 rz 180 deg; joints [-164.468, -66.384, -81.644, 18.14, 59.325, -9.489]
  Call Extruder(2565.60358)
  MoveL 203 to (41.51, -9.47, 15) mm, rotated rx -180 ry 0 rz 180 deg; joints [-163.355, -66.678, -80.65, 19.553, 58.855, -10.409]
  Call Extruder(2580.49946)
  MoveL 204 to (42.57, 0, 15) mm, rotated rx -180 ry 0 rz 180 deg; joints [-162.12, -66.888, -79.953, 21.075, 58.631, -11.343]
  Call Extruder(2595.39533)
  MoveL 205 to (41.5, 9.47, 15) mm, rotated rx -180 ry 0 rz 180 deg; joints [-160.81, -66.999, -79.588, 22.634, 58.663, -12.235]
  Call Extruder(2610.29099)
  MoveL 206 to (38.36, 18.47, 15) mm, rotated rx 180 ry 0 rz 180 deg; joints [-159.475, -67.004, -79.57, 24.16, 58.944, -13.03]
  Call Extruder(2625.18684)
  MoveL 207 to (33.29, 26.54, 15) mm, rotated rx -180 ry 0 rz 180 deg; joints [-158.16, -66.903, -79.902, 25.591, 59.456, -13.679]
  Call Extruder(2640.08266)
  MoveL 208 to (26.54, 33.28, 15) mm, rotated rx 180 ry 0 rz 180 deg; joints [-156.916, -66.703, -80.567, 26.869, 60.172, -14.144]
  Call Extruder(2654.97850)
  MoveL 209 to (18.47, 38.36, 15) mm, rotated rx 180 ry 0 rz -180 deg; joints [-155.789, -66.416, -81.533, 27.946, 61.054, -14.4]
  Call Extruder(2669.87417)
  MoveL 210 to (9.47, 41.51, 15) mm, rotated rx -180 ry 0 rz 180 deg; joints [-154.828, -66.063, -82.757, 28.781, 62.059, -14.434]
  Call Extruder(2684.77004)
  MoveL 211 to (0, 42.57, 15) mm, rotated rx -180 ry 0 rz 180 deg; joints [-154.081, -65.666, -84.179, 29.338, 63.14, -14.249]
  Call Extruder(2699.66591)
  MoveL 212 to (-9.47, 41.51, 15) mm, rotated rx 180 ry 0 rz 180 deg; joints [-153.594, -65.249, -85.733, 29.588, 64.248, -13.858]
  Call Extruder(2714.56156)
  MoveL 213 to (-18.47, 38.36, 15) mm, rotated rx -180 ry 0 rz -180 deg; joints [-153.408, -64.837, -87.344, 29.51, 65.335, -13.289]
  Call Extruder(2729.45742)
  MoveL 214 to (-26.54, 33.29, 15) mm, rotated rx -180 ry 0 rz 180 deg; joints [-153.557, -64.453, -88.933, 29.086, 66.352, -12.578]
  Call Extruder(2744.35323)
  MoveL 215 to (-33.28, 26.54, 15) mm, rotated rx 180 ry 0 rz 180 deg; joints [-154.059, -64.115, -90.42, 28.316, 67.254, -11.768]
  Call Extruder(2759.24908)
  MoveL 216 to (-38.36, 18.47, 15) mm, rotated rx -180 ry 0 rz 180 deg; joints [-154.913, -63.835, -91.729, 27.213, 67.996, -10.905]
  Call Extruder(2774.14474)
  MoveL 217 to (-41.51, 9.47, 15) mm, rotated rx 180 ry 0 rz 180 deg; joints [-156.091, -63.621, -92.787, 25.816, 68.538, -10.037]
  Call Extruder(2789.04062)
  MoveL 218 to (-42.57, 0, 15) mm, rotated rx 180 ry 0 rz -180 deg; joints [-157.533, -63.478, -93.535, 24.19, 68.846, -9.208]
  Call Extruder(2796.59489)
  MoveL 219 to (-42.03, -4.8, 15) mm, rotated rx 180 ry 0 rz 180 deg; joints [-158.35, -63.44, -93.741, 23.298, 68.871, -8.824]
  Set speed (130.0 mm/s)
  MoveL 220 to (-54.1, -7.67, 15) mm, rotated rx 180 ry 0 rz -180 deg; joints [-158.024, -63.107, -95.659, 23.409, 70.375, -8.273]
  Call Extruder(2800.66752)
  Set speed (30.0 mm/s)
  MoveL 221 to (-53.59, -12.23, 15) mm, rotated rx -180 ry 0 rz 180 deg; joints [-158.835, -63.077, -95.844, 22.535, 70.404, -7.923]
  Call Extruder(2811.59766)
  MoveL 222 to (-49.53, -23.85, 15) mm, rotated rx 180 ry 0 rz -180 deg; joints [-161.095, -63.073, -95.869, 20.152, 70.128, -7.111]
  Call Extruder(2822.52794)
  MoveL 223 to (-42.98, -34.27, 15) mm, rotated rx 180 ry 0 rz 180 deg; joints [-163.275, -63.149, -95.398, 17.893, 69.497, -6.452]
  Call Extruder(2833.45806)
  MoveL 224 to (-34.27, -42.98, 15) mm, rotated rx 180 ry 0 rz 180 deg; joints [-165.21, -63.31, -94.46, 15.919, 68.544, -5.956]
  Call Extruder(2844.38834)
  MoveL 225 to (-23.85, -49.53, 15) mm, rotated rx 180 ry 0 rz 180 deg; joints [-166.774, -63.558, -93.115, 14.357, 67.326, -5.635]
  Call Extruder(2855.31847)
  MoveL 226 to (-12.23, -53.59, 15) mm, rotated rx 180 ry 0 rz 180 deg; joints [-167.889, -63.895, -91.44, 13.286, 65.919, -5.503]
  Call Extruder(2866.24870)
  MoveL 227 to (0, -54.97, 15) mm, rotated rx 180 ry 0 rz 180 deg; joints [-168.526, -64.315, -89.529, 12.742, 64.405, -5.58]
  Call Extruder(2866.68050)
  MoveL 228 to (0.48, -54.91, 15) mm, rotated rx 180 ry 0 rz 180 deg; joints [-168.533, -64.333, -89.449, 12.741, 64.344, -5.591]
  Call Extruder(2877.17892)
  MoveL 229 to (12.23, -53.59, 15) mm, rotated rx 180 ry 0 rz 180 deg; joints [-168.697, -64.803, -87.483, 12.723, 62.868, -5.879]
  Call Extruder(2888.10906)
  MoveL 230 to (23.85, -49.53, 15) mm, rotated rx -180 ry 0 rz 180 deg; joints [-168.436, -65.336, -85.404, 13.199, 61.389, -6.408]
  Call Extruder(2899.03934)
  MoveL 231 to (34.27, -42.98, 15) mm, rotated rx 180 ry 0 rz 180 deg; joints [-167.797, -65.884, -83.393, 14.121, 60.043, -7.16]
  Call Extruder(2909.96946)
  MoveL 232 to (42.98, -34.27, 15) mm, rotated rx -180 ry 0 rz 180 deg; joints [-166.837, -66.413, -81.544, 15.424, 58.895, -8.112]
  Call Extruder(2920.89974)
  MoveL 233 to (49.53, -23.85, 15) mm, rotated rx 180 ry 0 rz 180 deg; joints [-165.618, -66.891, -79.944, 17.031, 58, -9.22]
  Call Extruder(2931.82988)
  MoveL 234 to (53.59, -12.23, 15) mm, rotated rx -180 ry 0 rz -180 deg; joints [-164.2, -67.283, -78.667, 18.856, 57.4, -10.426]
  Call Extruder(2942.76010)
  MoveL 235 to (54.97, 0, 15) mm, rotated rx -180 ry 0 rz 180 deg; joints [-162.641, -67.564, -77.772, 20.81, 57.122, -11.658]
  Call Extruder(2953.69032)
  MoveL 236 to (53.59, 12.23, 15) mm, rotated rx 180 ry 0 rz 180 deg; joints [-160.996, -67.713, -77.302, 22.8, 57.173, -12.837]
  Call Extruder(2964.62046)
  MoveL 237 to (49.52, 23.85, 15) mm, rotated rx 180 ry 0 rz -180 deg; joints [-159.322, -67.721, -77.28, 24.738, 57.546, -13.888]
  Call Extruder(2975.55074)
  MoveL 238 to (42.98, 34.27, 15) mm, rotated rx 180 ry 0 rz 180 deg; joints [-157.673, -67.585, -77.706, 26.546, 58.216, -14.743]
  Call Extruder(2986.48086)
  MoveL 239 to (34.27, 42.98, 15) mm, rotated rx 180 ry 0 rz 180 deg; joints [-156.102, -67.316, -78.56, 28.158, 59.144, -15.351]
  Call Extruder(2997.41114)
  MoveL 240 to (23.85, 49.52, 15) mm, rotated rx -180 ry 0 rz 180 deg; joints [-154.667, -66.934, -79.801, 29.517, 60.28, -15.679]
  Call Extruder(3008.34128)
  MoveL 241 to (12.23, 53.59, 15) mm, rotated rx 180 ry 0 rz 180 deg; joints [-153.426, -66.464, -81.373, 30.578, 61.569, -15.712]
  Call Extruder(3019.27150)
  MoveL 242 to (0, 54.97, 15) mm, rotated rx 180 ry 0 rz -180 deg; joints [-152.438, -65.938, -83.2, 31.301, 62.951, -15.457]
  Call Extruder(3030.20173)
  MoveL 243 to (-12.23, 53.59, 15) mm, rotated rx -180 ry 0 rz 180 deg; joints [-151.764, -65.39, -85.2, 31.652, 64.366, -14.933]
  Call Extruder(3041.13186)
  MoveL 244 to (-23.85, 49.52, 15) mm, rotated rx -180 ry 0 rz 180 deg; joints [-151.463, -64.854, -87.276, 31.597, 65.753, -14.177]
  Call Extruder(3052.06214)
  MoveL 245 to (-34.27, 42.98, 15) mm, rotated rx 180 ry 0 rz 180 deg; joints [-151.589, -64.361, -89.33, 31.109, 67.056, -13.238]
  Call Extruder(3062.99226)
  MoveL 246 to (-42.98, 34.27, 15) mm, rotated rx -180 ry 0 rz -180 deg; joints [-152.179, -63.933, -91.259, 30.171, 68.218, -12.174]
  Call Extruder(3073.92254)
  MoveL 247 to (-49.52, 23.85, 15) mm, rotated rx 180 ry 0 rz 180 deg; joints [-153.248, -63.587, -92.962, 28.788, 69.184, -11.049]
  Call Extruder(3084.85268)
  MoveL 248 to (-53.59, 12.23, 15) mm, rotated rx 180 ry 0 rz 180 deg; joints [-154.769, -63.33, -94.344, 26.995, 69.902, -9.929]
  Call Extruder(3095.78291)
  MoveL 249 to (-54.97, 0, 15) mm, rotated rx 180 ry 0 rz -180 deg; joints [-156.673, -63.162, -95.325, 24.869, 70.321, -8.872]
  Call Extruder(3101.30852)
  MoveL 250 to (-54.27, -6.18, 15) mm, rotated rx -180 ry 0 rz -180 deg; joints [-157.76, -63.117, -95.597, 23.694, 70.365, -8.389]
  Set speed (130.0 mm/s)
  MoveL 251 to (-49.9, -9.51, 15) mm, rotated rx -180 ry 0 rz 180 deg; joints [-158.616, -63.189, -95.158, 22.845, 69.905, -8.236]
  MoveL 252 to (-13.82, -4.92, 15) mm, rotated rx -180 ry 0 rz 180 deg; joints [-160.062, -64.324, -89.488, 22.01, 65.489, -9.52]
  Call Extruder(3134.48354)
  Set speed (20.0 mm/s)
  MoveL 253 to (-4.92, -13.82, 15) mm, rotated rx -180 ry 0 rz 180 deg; joints [-161.89, -64.538, -88.572, 20.137, 64.541, -8.957]
  Call Extruder(3204.29014)
  MoveL 254 to (13.82, 4.91, 15) mm, rotated rx -180 ry 0 rz -180 deg; joints [-160.09, -65.574, -84.517, 22.678, 62.042, -11.084]
  Call Extruder(3237.46517)
  MoveL 255 to (4.92, 13.82, 15) mm, rotated rx 180 ry 0 rz -180 deg; joints [-158.352, -65.334, -85.411, 24.461, 62.985, -11.675]
  Set speed (130.0 mm/s)
  MoveL 256 to (4.91, 13.82, 20) mm, rotated rx -180 ry 0 rz -180 deg; joints [-158.352, -64.575, -85.875, 24.524, 62.716, -11.813]
  MoveL 257 to (-26.25, -4.54, 20) mm, rotated rx 180 ry 0 rz 180 deg; joints [-159.288, -63.118, -91.846, 22.651, 66.682, -9.38]
  Call Extruder(3239.69780)
  Set speed (60.0 mm/s)
  MoveL 258 to (-26.09, -5.96, 20) mm, rotated rx -180 ry 0 rz 180 deg; joints [-159.522, -63.106, -91.903, 22.393, 66.686, -9.262]
  Call Extruder(3249.06259)
  MoveL 259 to (-24.12, -11.61, 20) mm, rotated rx -180 ry 0 rz -180 deg; joints [-160.532, -63.103, -91.915, 21.305, 66.535, -8.827]
  Call Extruder(3258.42751)
  MoveL 260 to (-20.93, -16.69, 20) mm, rotated rx -180 ry 0 rz -180 deg; joints [-161.513, -63.152, -91.693, 20.273, 66.226, -8.47]
  Call Extruder(3267.79271)
  MoveL 261 to (-16.69, -20.93, 20) mm, rotated rx -180 ry 0 rz 180 deg; joints [-162.406, -63.249, -91.251, 19.358, 65.771, -8.204]
  Call Extruder(3277.15764)
  MoveL 262 to (-11.61, -24.12, 20) mm, rotated rx 180 ry 0 rz 180 deg; joints [-163.159, -63.393, -90.611, 18.612, 65.196, -8.041]
  Call Extruder(3286.52242)
  MoveL 263 to (-5.96, -26.09, 20) mm, rotated rx 180 ry 0 rz 180 deg; joints [-163.733, -63.579, -89.809, 18.075, 64.532, -7.989]
  Call Extruder(3295.88753)
  MoveL 264 to (0, -26.77, 20) mm, rotated rx 180 ry 0 rz 180 deg; joints [-164.103, -63.801, -88.888, 17.772, 63.814, -8.051]
  Call Extruder(3305.25263)
  MoveL 265 to (5.96, -26.09, 20) mm, rotated rx 180 ry 0 rz 180 deg; joints [-164.258, -64.048, -87.893, 17.715, 63.081, -8.229]
  Call Extruder(3314.61744)
  MoveL 266 to (11.61, -24.11, 20) mm, rotated rx 180 ry 0 rz 180 deg; joints [-164.201, -64.309, -86.877, 17.897, 62.37, -8.518]
  Call Extruder(3323.98235)
  MoveL 267 to (16.69, -20.93, 20) mm, rotated rx 180 ry 0 rz 180 deg; joints [-163.944, -64.571, -85.889, 18.305, 61.719, -8.908]
  Call Extruder(3333.34755)
  MoveL 268 to (20.93, -16.69, 20) mm, rotated rx -180 ry 0 rz 180 deg; joints [-163.508, -64.819, -84.978, 18.91, 61.161, -9.383]
  Call Extruder(3342.71248)
  MoveL 269 to (24.12, -11.61, 20) mm, rotated rx 180 ry 0 rz 180 deg; joints [-162.92, -65.04, -84.188, 19.678, 60.721, -9.92]
  Call Extruder(3352.07727)
  MoveL 270 to (26.09, -5.96, 20) mm, rotated rx -180 ry 0 rz -180 deg; joints [-162.209, -65.219, -83.557, 20.568, 60.423, -10.493]
  Call Extruder(3361.44237)
  MoveL 271 to (26.77, 0, 20) mm, rotated rx 180 ry 0 rz -180 deg; joints [-161.41, -65.346, -83.115, 21.536, 60.279, -11.07]
  Call Extruder(3370.80747)
  MoveL 272 to (26.09, 5.96, 20) mm, rotated rx -180 ry 0 rz 180 deg; joints [-160.556, -65.414, -82.883, 22.535, 60.294, -11.619]
  Call Extruder(3380.17228)
  MoveL 273 to (24.11, 11.61, 20) mm, rotated rx 180 ry 0 rz 180 deg; joints [-159.683, -65.417, -82.872, 23.52, 60.466, -12.109]
  Call Extruder(3389.53719)
  MoveL 274 to (20.93, 16.69, 20) mm, rotated rx -180 ry 0 rz 180 deg; joints [-158.826, -65.356, -83.082, 24.447, 60.786, -12.51]
  Call Extruder(3398.90240)
  MoveL 275 to (16.69, 20.93, 20) mm, rotated rx -180 ry 0 rz 180 deg; joints [-158.019, -65.234, -83.505, 25.276, 61.235, -12.802]
  Call Extruder(3408.26731)
  MoveL 276 to (11.61, 24.11, 20) mm, rotated rx 180 ry 0 rz 180 deg; joints [-157.299, -65.06, -84.118, 25.972, 61.791, -12.967]
  Call Extruder(3417.63211)
  MoveL 277 to (5.96, 26.09, 20) mm, rotated rx -180 ry 0 rz 180 deg; joints [-156.697, -64.843, -84.894, 26.505, 62.428, -12.998]
  Call Extruder(3426.99722)
  MoveL 278 to (0, 26.77, 20) mm, rotated rx 180 ry 0 rz 180 deg; joints [-156.245, -64.596, -85.795, 26.85, 63.114, -12.894]
  Call Extruder(3436.36232)
  MoveL 279 to (-5.96, 26.09, 20) mm, rotated rx 180 ry 0 rz 180 deg; joints [-155.969, -64.335, -86.777, 26.987, 63.818, -12.663]
  Call Extruder(3445.72711)
  MoveL 280 to (-11.61, 24.11, 20) mm, rotated rx -180 ry 0 rz 180 deg; joints [-155.891, -64.073, -87.793, 26.906, 64.507, -12.321]
  Call Extruder(3455.09203)
  MoveL 281 to (-16.69, 20.93, 20) mm, rotated rx 180 ry 0 rz -180 deg; joints [-156.025, -63.824, -88.791, 26.603, 65.148, -11.887]
  Call Extruder(3464.45724)
  MoveL 282 to (-20.93, 16.69, 20) mm, rotated rx 180 ry 0 rz 180 deg; joints [-156.374, -63.6, -89.723, 26.084, 65.711, -11.385]
  Call Extruder(3473.82215)
  MoveL 283 to (-24.11, 11.61, 20) mm, rotated rx 180 ry 0 rz 180 deg; joints [-156.928, -63.41, -90.538, 25.367, 66.168, -10.845]
  Call Extruder(3483.18695)
  MoveL 284 to (-26.09, 5.96, 20) mm, rotated rx 180 ry 0 rz -180 deg; joints [-157.665, -63.261, -91.195, 24.482, 66.494, -10.294]
  Call Extruder(3492.55206)
  MoveL 285 to (-26.77, 0, 20) mm, rotated rx -180 ry 0 rz 180 deg; joints [-158.546, -63.159, -91.659, 23.473, 66.671, -9.758]
  Call Extruder(3497.34079)
  MoveL 286 to (-26.42, -3.05, 20) mm, rotated rx -180 ry 0 rz 180 deg; joints [-159.044, -63.131, -91.786, 22.922, 66.679, -9.503]
  Set speed (130.0 mm/s)
  MoveL 287 to (-41.86, -6.29, 20) mm, rotated rx 180 ry 0 rz 180 deg; joints [-158.606, -62.623, -94.282, 23.07, 68.578, -8.842]
  Call Extruder(3502.33864)
  Set speed (60.0 mm/s)
  MoveL 288 to (-41.51, -9.47, 20) mm, rotated rx 180 ry 0 rz 180 deg; joints [-159.151, -62.599, -94.41, 22.475, 68.591, -8.587]
  Call Extruder(3517.23429)
  MoveL 289 to (-38.36, -18.47, 20) mm, rotated rx 180 ry 0 rz 180 deg; joints [-160.835, -62.595, -94.429, 20.681, 68.363, -7.924]
  Call Extruder(3532.13014)
  MoveL 290 to (-33.29, -26.54, 20) mm, rotated rx -180 ry 0 rz 180 deg; joints [-162.466, -62.663, -94.069, 18.98, 67.872, -7.381]
  Call Extruder(3547.02596)
  MoveL 291 to (-26.54, -33.28, 20) mm, rotated rx -180 ry 0 rz -180 deg; joints [-163.93, -62.804, -93.352, 17.482, 67.142, -6.975]
  Call Extruder(3561.92181)
  MoveL 292 to (-18.47, -38.36, 20) mm, rotated rx 180 ry 0 rz 180 deg; joints [-165.137, -63.017, -92.32, 16.28, 66.214, -6.718]
  Call Extruder(3576.81746)
  MoveL 293 to (-9.47, -41.51, 20) mm, rotated rx -180 ry 0 rz 180 deg; joints [-166.024, -63.298, -91.031, 15.437, 65.141, -6.621]
  Call Extruder(3591.71334)
  MoveL 294 to (0, -42.57, 20) mm, rotated rx -180 ry 0 rz -180 deg; joints [-166.562, -63.639, -89.555, 14.987, 63.984, -6.697]
  Call Extruder(3606.60921)
  MoveL 295 to (9.47, -41.51, 20) mm, rotated rx -180 ry 0 rz 180 deg; joints [-166.745, -64.028, -87.97, 14.938, 62.807, -6.951]
  Call Extruder(3621.50487)
  MoveL 296 to (18.47, -38.36, 20) mm, rotated rx 180 ry 0 rz 180 deg; joints [-166.591, -64.446, -86.355, 15.275, 61.671, -7.384]
  Call Extruder(3636.40072)
  MoveL 297 to (26.54, -33.29, 20) mm, rotated rx 180 ry 0 rz 180 deg; joints [-166.133, -64.871, -84.791, 15.963, 60.635, -7.985]
  Call Extruder(3651.29654)
  MoveL 298 to (33.29, -26.54, 20) mm, rotated rx 180 ry 0 rz 180 deg; joints [-165.409, -65.278, -83.351, 16.955, 59.749, -8.732]
  Call Extruder(3666.19239)
  MoveL 299 to (38.36, -18.47, 20) mm, rotated rx 180 ry 0 rz 180 deg; joints [-164.468, -65.642, -82.104, 18.193, 59.058, -9.591]
  Call Extruder(3681.08804)
  MoveL 300 to (41.51, -9.47, 20) mm, rotated rx 180 ry 0 rz 180 deg; joints [-163.355, -65.94, -81.109, 19.61, 58.593, -10.518]
  Call Extruder(3695.98391)
  MoveL 301 to (42.57, 0, 20) mm, rotated rx -180 ry 0 rz 180 deg; joints [-162.12, -66.153, -80.412, 21.136, 58.374, -11.459]
  Call Extruder(3710.87979)
  MoveL 302 to (41.5, 9.47, 20) mm, rotated rx 180 ry 0 rz 180 deg; joints [-160.81, -66.266, -80.047, 22.698, 58.41, -12.359]
  Call Extruder(3725.77545)
  MoveL 303 to (38.36, 18.47, 20) mm, rotated rx 180 ry 0 rz 180 deg; joints [-159.475, -66.271, -80.029, 24.228, 58.694, -13.161]
  Call Extruder(3740.67129)
  MoveL 304 to (33.29, 26.54, 20) mm, rotated rx 180 ry 0 rz 180 deg; joints [-158.16, -66.169, -80.361, 25.662, 59.208, -13.818]
  Call Extruder(3755.56712)
  MoveL 305 to (26.54, 33.28, 20) mm, rotated rx -180 ry 0 rz 180 deg; joints [-156.916, -65.966, -81.026, 26.942, 59.925, -14.289]
  Call Extruder(3770.46296)
  MoveL 306 to (18.47, 38.36, 20) mm, rotated rx 180 ry 0 rz -180 deg; joints [-155.789, -65.675, -81.994, 28.02, 60.806, -14.551]
  Call Extruder(3785.35862)
  MoveL 307 to (9.47, 41.51, 20) mm, rotated rx -180 ry 0 rz 180 deg; joints [-154.828, -65.317, -83.218, 28.854, 61.809, -14.59]
  Call Extruder(3800.25450)
  MoveL 308 to (0, 42.57, 20) mm, rotated rx 180 ry 0 rz 180 deg; joints [-154.081, -64.913, -84.641, 29.411, 62.886, -14.409]
  Call Extruder(3815.15037)
  MoveL 309 to (-9.47, 41.51, 20) mm, rotated rx 180 ry 0 rz 180 deg; joints [-153.594, -64.489, -86.197, 29.66, 63.99, -14.021]
  Call Extruder(3830.04602)
  MoveL 310 to (-18.47, 38.36, 20) mm, rotated rx -180 ry 0 rz -180 deg; joints [-153.408, -64.069, -87.81, 29.578, 65.072, -13.454]
  Call Extruder(3844.94187)
  MoveL 311 to (-26.54, 33.29, 20) mm, rotated rx 180 ry 0 rz 180 deg; joints [-153.557, -63.676, -89.401, 29.152, 66.083, -12.742]
  Call Extruder(3859.83769)
  MoveL 312 to (-33.28, 26.54, 20) mm, rotated rx 180 ry 0 rz -180 deg; joints [-154.059, -63.329, -90.891, 28.379, 66.978, -11.93]
  Call Extruder(3874.73354)
  MoveL 313 to (-38.36, 18.47, 20) mm, rotated rx 180 ry 0 rz 180 deg; joints [-154.913, -63.042, -92.202, 27.273, 67.713, -11.063]
  Call Extruder(3889.62920)
  MoveL 314 to (-41.5, 9.47, 20) mm, rotated rx -180 ry 0 rz 180 deg; joints [-156.091, -62.822, -93.263, 25.872, 68.248, -10.189]
  Call Extruder(3904.52507)
  MoveL 315 to (-42.57, 0, 20) mm, rotated rx 180 ry 0 rz -180 deg; joints [-157.533, -62.674, -94.013, 24.242, 68.549, -9.352]
  Call Extruder(3912.07935)
  MoveL 316 to (-42.03, -4.8, 20) mm, rotated rx 180 ry 0 rz 180 deg; joints [-158.35, -62.635, -94.22, 23.349, 68.571, -8.962]
  Set speed (130.0 mm/s)
  MoveL 317 to (-54.1, -7.67, 20) mm, rotated rx 180 ry 0 rz -180 deg; joints [-158.024, -62.289, -96.143, 23.457, 70.069, -8.414]
  Call Extruder(3916.15198)
  Set speed (30.0 mm/s)
  MoveL 318 to (-53.59, -12.23, 20) mm, rotated rx -180 ry 0 rz 180 deg; joints [-158.835, -62.258, -96.328, 22.581, 70.095, -8.059]
  Call Extruder(3927.08211)
  MoveL 319 to (-49.53, -23.85, 20) mm, rotated rx 180 ry 0 rz 180 deg; joints [-161.095, -62.254, -96.353, 20.194, 69.813, -7.234]
  Call Extruder(3938.01240)
  MoveL 320 to (-42.98, -34.27, 20) mm, rotated rx -180 ry 0 rz 180 deg; joints [-163.275, -62.334, -95.881, 17.932, 69.18, -6.561]
  Call Extruder(3948.94251)
  MoveL 321 to (-34.27, -42.98, 20) mm, rotated rx 180 ry 0 rz 180 deg; joints [-165.21, -62.5, -94.941, 15.955, 68.227, -6.053]
  Call Extruder(3959.87280)
  MoveL 322 to (-23.85, -49.52, 20) mm, rotated rx 180 ry 0 rz 180 deg; joints [-166.774, -62.757, -93.592, 14.391, 67.012, -5.722]
  Call Extruder(3970.80293)
  MoveL 323 to (-12.23, -53.59, 20) mm, rotated rx 180 ry 0 rz 180 deg; joints [-167.889, -63.104, -91.913, 13.319, 65.61, -5.584]
  Call Extruder(3981.73315)
  MoveL 324 to (0, -54.97, 20) mm, rotated rx 180 ry 0 rz 180 deg; joints [-168.526, -63.535, -89.998, 12.775, 64.102, -5.656]
  Call Extruder(3982.53779)
  MoveL 325 to (0.9, -54.87, 20) mm, rotated rx 180 ry 0 rz -180 deg; joints [-168.539, -63.57, -89.849, 12.773, 63.989, -5.678]
  Call Extruder(3992.66338)
  MoveL 326 to (12.23, -53.59, 20) mm, rotated rx 180 ry 0 rz 180 deg; joints [-168.697, -64.034, -87.949, 12.757, 62.572, -5.954]
  Call Extruder(4003.59352)
  MoveL 327 to (23.85, -49.53, 20) mm, rotated rx -180 ry 0 rz 180 deg; joints [-168.436, -64.577, -85.867, 13.236, 61.101, -6.485]
  Call Extruder(4014.52380)
  MoveL 328 to (34.27, -42.98, 20) mm, rotated rx 180 ry 0 rz 180 deg; joints [-167.797, -65.134, -83.854, 14.162, 59.764, -7.242]
  Call Extruder(4025.45392)
  MoveL 329 to (42.98, -34.27, 20) mm, rotated rx 180 ry 0 rz 180 deg; joints [-166.837, -65.672, -82.004, 15.469, 58.624, -8.199]
  Call Extruder(4036.38420)
  MoveL 330 to (49.52, -23.85, 20) mm, rotated rx -180 ry 0 rz 180 deg; joints [-165.618, -66.156, -80.403, 17.081, 57.737, -9.315]
  Call Extruder(4047.31433)
  MoveL 331 to (53.59, -12.23, 20) mm, rotated rx -180 ry 0 rz -180 deg; joints [-164.2, -66.554, -79.125, 18.913, 57.144, -10.53]
  Call Extruder(4058.24456)
  MoveL 332 to (54.97, 0, 20) mm, rotated rx 180 ry 0 rz 180 deg; joints [-162.641, -66.838, -78.231, 20.872, 56.872, -11.771]
  Call Extruder(4069.17478)
  MoveL 333 to (53.59, 12.23, 20) mm, rotated rx -180 ry 0 rz 180 deg; joints [-160.996, -66.989, -77.761, 22.867, 56.928, -12.96]
  Call Extruder(4080.10492)
  MoveL 334 to (49.53, 23.85, 20) mm, rotated rx -180 ry 0 rz -180 deg; joints [-159.322, -66.996, -77.739, 24.809, 57.305, -14.02]
  Call Extruder(4091.03520)
  MoveL 335 to (42.98, 34.27, 20) mm, rotated rx 180 ry 0 rz 180 deg; joints [-157.673, -66.859, -78.165, 26.621, 57.977, -14.884]
  Call Extruder(4101.96532)
  MoveL 336 to (34.27, 42.98, 20) mm, rotated rx 180 ry 0 rz 180 deg; joints [-156.102, -66.587, -79.019, 28.234, 58.905, -15.5]
  Call Extruder(4112.89560)
  MoveL 337 to (23.85, 49.52, 20) mm, rotated rx -180 ry 0 rz 180 deg; joints [-154.667, -66.2, -80.261, 29.595, 60.041, -15.835]
  Call Extruder(4123.82574)
  MoveL 338 to (12.23, 53.59, 20) mm, rotated rx 180 ry 0 rz 180 deg; joints [-153.426, -65.723, -81.833, 30.656, 61.327, -15.875]
  Call Extruder(4134.75596)
  MoveL 339 to (0, 54.97, 20) mm, rotated rx 180 ry 0 rz 180 deg; joints [-152.438, -65.189, -83.662, 31.378, 62.706, -15.624]
  Call Extruder(4145.68618)
  MoveL 340 to (-12.23, 53.59, 20) mm, rotated rx 180 ry 0 rz 180 deg; joints [-151.764, -64.632, -85.663, 31.727, 64.115, -15.105]
  Call Extruder(4156.61632)
  MoveL 341 to (-23.85, 49.52, 20) mm, rotated rx -180 ry 0 rz 180 deg; joints [-151.463, -64.086, -87.742, 31.669, 65.496, -14.351]
  Call Extruder(4167.54660)
  MoveL 342 to (-34.27, 42.98, 20) mm, rotated rx -180 ry 0 rz 180 deg; joints [-151.589, -63.582, -89.799, 31.177, 66.791, -13.412]
  Call Extruder(4178.47672)
  MoveL 343 to (-42.98, 34.27, 20) mm, rotated rx 180 ry 0 rz -180 deg; joints [-152.179, -63.143, -91.732, 30.236, 67.944, -12.346]
  Call Extruder(4189.40700)
  MoveL 344 to (-49.52, 23.85, 20) mm, rotated rx -180 ry 0 rz 180 deg; joints [-153.248, -62.787, -93.438, 28.848, 68.901, -11.216]
  Call Extruder(4200.33714)
  MoveL 345 to (-53.59, 12.23, 20) mm, rotated rx 180 ry 0 rz -180 deg; joints [-154.769, -62.521, -94.824, 27.05, 69.609, -10.088]
  Call Extruder(4211.26736)
  MoveL 346 to (-54.97, 0, 20) mm, rotated rx 180 ry 0 rz -180 deg; joints [-156.673, -62.346, -95.807, 24.92, 70.02, -9.021]
  Call Extruder(4216.79298)
  MoveL 347 to (-54.27, -6.18, 20) mm, rotated rx 180 ry 0 rz 180 deg; joints [-157.76, -62.3, -96.08, 23.742, 70.06, -8.531]
  Set speed (130.0 mm/s)
  MoveL 348 to (-49.9, -9.51, 20) mm, rotated rx -180 ry 0 rz 180 deg; joints [-158.616, -62.375, -95.641, 22.893, 69.6, -8.373]
  MoveL 349 to (-4.92, 13.82, 20) mm, rotated rx 180 ry 0 rz 180 deg; joints [-157.786, -64.164, -87.435, 24.903, 63.875, -11.553]
  Call Extruder(4249.96799)
  Set speed (20.0 mm/s)
  MoveL 350 to (-13.82, 4.91, 20) mm, rotated rx -180 ry 0 rz 180 deg; joints [-158.572, -63.681, -89.381, 23.76, 65.057, -10.517]
  Call Extruder(4319.77461)
  MoveL 351 to (4.92, -13.82, 20) mm, rotated rx 180 ry 0 rz 180 deg; joints [-162.368, -64.157, -87.465, 19.862, 63.066, -9.293]
  Call Extruder(4352.94962)
  MoveL 352 to (13.82, -4.91, 20) mm, rotated rx 180 ry 0 rz 180 deg; joints [-161.491, -64.665, -85.541, 21.095, 61.889, -10.302]
  Set speed (130.0 mm/s)
  MoveL 353 to (13.82, -4.92, 25) mm, rotated rx 180 ry 0 rz 180 deg; joints [-161.491, -63.908, -85.995, 21.154, 61.607, -10.426]
  MoveL 354 to (-26.25, -4.54, 25) mm, rotated rx 180 ry 0 rz 180 deg; joints [-159.288, -62.327, -92.311, 22.706, 66.381, -9.517]
  Call Extruder(4355.18225)
  Set speed (60.0 mm/s)
  MoveL 355 to (-26.09, -5.96, 25) mm, rotated rx -180 ry 0 rz 180 deg; joints [-159.522, -62.314, -92.368, 22.447, 66.383, -9.398]
  Call Extruder(4364.54704)
  MoveL 356 to (-24.11, -11.61, 25) mm, rotated rx 180 ry 0 rz 180 deg; joints [-160.532, -62.312, -92.379, 21.357, 66.231, -8.957]
  Call Extruder(4373.91195)
  MoveL 357 to (-20.93, -16.69, 25) mm, rotated rx -180 ry 0 rz 180 deg; joints [-161.513, -62.361, -92.157, 20.323, 65.919, -8.593]
  Call Extruder(4383.27716)
  MoveL 358 to (-16.69, -20.93, 25) mm, rotated rx 180 ry 0 rz 180 deg; joints [-162.406, -62.461, -91.714, 19.406, 65.465, -8.322]
  Call Extruder(4392.64208)
  MoveL 359 to (-11.61, -24.12, 25) mm, rotated rx -180 ry 0 rz 180 deg; joints [-163.159, -62.609, -91.073, 18.659, 64.891, -8.155]
  Call Extruder(4402.00687)
  MoveL 360 to (-5.96, -26.09, 25) mm, rotated rx 180 ry 0 rz 180 deg; joints [-163.733, -62.8, -90.27, 18.122, 64.229, -8.099]
  Call Extruder(4411.37197)
  MoveL 361 to (0, -26.77, 25) mm, rotated rx 180 ry 0 rz 180 deg; joints [-164.103, -63.026, -89.346, 17.82, 63.514, -8.158]
  Call Extruder(4420.73709)
  MoveL 362 to (5.96, -26.09, 25) mm, rotated rx 180 ry 0 rz 180 deg; joints [-164.258, -63.279, -88.351, 17.763, 62.784, -8.335]
  Call Extruder(4430.10188)
  MoveL 363 to (11.61, -24.11, 25) mm, rotated rx 180 ry 0 rz 180 deg; joints [-164.201, -63.545, -87.333, 17.947, 62.077, -8.625]
  Call Extruder(4439.46679)
  MoveL 364 to (16.69, -20.93, 25) mm, rotated rx -180 ry 0 rz 180 deg; joints [-163.944, -63.812, -86.344, 18.356, 61.431, -9.017]
  Call Extruder(4448.83200)
  MoveL 365 to (20.93, -16.69, 25) mm, rotated rx 180 ry 0 rz 180 deg; joints [-163.508, -64.065, -85.432, 18.964, 60.876, -9.494]
  Call Extruder(4458.19692)
  MoveL 366 to (24.12, -11.61, 25) mm, rotated rx 180 ry 0 rz 180 deg; joints [-162.92, -64.289, -84.641, 19.734, 60.441, -10.036]
  Call Extruder(4467.56172)
  MoveL 367 to (26.09, -5.96, 25) mm, rotated rx -180 ry 0 rz -180 deg; joints [-162.209, -64.472, -84.009, 20.627, 60.147, -10.613]
  Call Extruder(4476.92682)
  MoveL 368 to (26.77, 0, 25) mm, rotated rx 180 ry 0 rz -180 deg; joints [-161.41, -64.601, -83.567, 21.598, 60.006, -11.195]
  Call Extruder(4486.29192)
  MoveL 369 to (26.09, 5.96, 25) mm, rotated rx -180 ry 0 rz 180 deg; joints [-160.556, -64.669, -83.334, 22.599, 60.024, -11.749]
  Call Extruder(4495.65673)
  MoveL 370 to (24.11, 11.61, 25) mm, rotated rx 180 ry 0 rz -180 deg; joints [-159.683, -64.673, -83.323, 23.586, 60.198, -12.243]
  Call Extruder(4505.02164)
  MoveL 371 to (20.93, 16.69, 25) mm, rotated rx 180 ry 0 rz 180 deg; joints [-158.826, -64.611, -83.534, 24.515, 60.518, -12.65]
  Call Extruder(4514.38685)
  MoveL 372 to (16.69, 20.93, 25) mm, rotated rx -180 ry 0 rz 180 deg; joints [-158.019, -64.487, -83.957, 25.346, 60.968, -12.946]
  Call Extruder(4523.75176)
  MoveL 373 to (11.61, 24.11, 25) mm, rotated rx -180 ry 0 rz 180 deg; joints [-157.299, -64.31, -84.571, 26.043, 61.524, -13.115]
  Call Extruder(4533.11656)
  MoveL 374 to (5.96, 26.09, 25) mm, rotated rx -180 ry 0 rz 180 deg; joints [-156.697, -64.089, -85.347, 26.575, 62.159, -13.149]
  Call Extruder(4542.48166)
  MoveL 375 to (0, 26.77, 25) mm, rotated rx 180 ry 0 rz 180 deg; joints [-156.245, -63.838, -86.249, 26.92, 62.843, -13.048]
  Call Extruder(4551.84677)
  MoveL 376 to (-5.96, 26.09, 25) mm, rotated rx 180 ry 0 rz 180 deg; joints [-155.969, -63.572, -87.233, 27.056, 63.544, -12.819]
  Call Extruder(4561.21156)
  MoveL 377 to (-11.61, 24.12, 25) mm, rotated rx 180 ry 0 rz 180 deg; joints [-155.891, -63.305, -88.25, 26.974, 64.229, -12.477]
  Call Extruder(4570.57648)
  MoveL 378 to (-16.69, 20.93, 25) mm, rotated rx 180 ry 0 rz -180 deg; joints [-156.025, -63.05, -89.25, 26.669, 64.866, -12.042]
  Call Extruder(4579.94169)
  MoveL 379 to (-20.93, 16.69, 25) mm, rotated rx -180 ry 0 rz 180 deg; joints [-156.374, -62.821, -90.183, 26.148, 65.425, -11.54]
  Call Extruder(4589.30660)
  MoveL 380 to (-24.11, 11.61, 25) mm, rotated rx 180 ry 0 rz 180 deg; joints [-156.928, -62.626, -91, 25.429, 65.877, -10.996]
  Call Extruder(4598.67140)
  MoveL 381 to (-26.09, 5.96, 25) mm, rotated rx 180 ry 0 rz 180 deg; joints [-157.665, -62.474, -91.658, 24.541, 66.199, -10.441]
  Call Extruder(4608.03651)
  MoveL 382 to (-26.77, 0, 25) mm, rotated rx 180 ry 0 rz 180 deg; joints [-158.546, -62.369, -92.123, 23.529, 66.371, -9.9]
  Call Extruder(4612.82524)
  MoveL 383 to (-26.42, -3.05, 25) mm, rotated rx 180 ry 0 rz 180 deg; joints [-159.044, -62.34, -92.25, 22.977, 66.378, -9.642]
  Set speed (130.0 mm/s)
  MoveL 384 to (-41.86, -6.3, 25) mm, rotated rx -180 ry 0 rz 180 deg; joints [-158.606, -61.816, -94.751, 23.122, 68.268, -8.984]
  Call Extruder(4617.82309)
  Set speed (60.0 mm/s)
  MoveL 385 to (-41.5, -9.47, 25) mm, rotated rx 180 ry 0 rz 180 deg; joints [-159.151, -61.791, -94.88, 22.526, 68.279, -8.726]
  Call Extruder(4632.71874)
  MoveL 386 to (-38.36, -18.47, 25) mm, rotated rx 180 ry 0 rz -180 deg; joints [-160.835, -61.787, -94.899, 20.729, 68.048, -8.052]
  Call Extruder(4647.61459)
  MoveL 387 to (-33.29, -26.54, 25) mm, rotated rx -180 ry 0 rz 180 deg; joints [-162.466, -61.858, -94.538, 19.024, 67.555, -7.5]
  Call Extruder(4662.51040)
  MoveL 388 to (-26.54, -33.28, 25) mm, rotated rx 180 ry 0 rz -180 deg; joints [-163.93, -62.004, -93.82, 17.524, 66.825, -7.084]
  Call Extruder(4677.40626)
  MoveL 389 to (-18.47, -38.36, 25) mm, rotated rx 180 ry 0 rz 180 deg; joints [-165.137, -62.223, -92.785, 16.321, 65.898, -6.819]
  Call Extruder(4692.30191)
  MoveL 390 to (-9.47, -41.51, 25) mm, rotated rx -180 ry 0 rz -180 deg; joints [-166.024, -62.512, -91.493, 15.477, 64.829, -6.717]
  Call Extruder(4707.19778)
  MoveL 391 to (0, -42.57, 25) mm, rotated rx -180 ry 0 rz 180 deg; joints [-166.562, -62.861, -90.015, 15.027, 63.677, -6.789]
  Call Extruder(4722.09366)
  MoveL 392 to (9.47, -41.51, 25) mm, rotated rx 180 ry 0 rz 180 deg; joints [-166.745, -63.259, -88.427, 14.98, 62.506, -7.042]
  Call Extruder(4736.98932)
  MoveL 393 to (18.47, -38.36, 25) mm, rotated rx -180 ry 0 rz 180 deg; joints [-166.591, -63.686, -86.81, 15.318, 61.376, -7.476]
  Call Extruder(4751.88516)
  MoveL 394 to (26.54, -33.28, 25) mm, rotated rx 180 ry 0 rz -180 deg; joints [-166.133, -64.118, -85.244, 16.01, 60.346, -8.08]
  Call Extruder(4766.78098)
  MoveL 395 to (33.29, -26.54, 25) mm, rotated rx 180 ry 0 rz 180 deg; joints [-165.409, -64.532, -83.803, 17.005, 59.468, -8.832]
  Call Extruder(4781.67684)
  MoveL 396 to (38.36, -18.47, 25) mm, rotated rx 180 ry 0 rz 180 deg; joints [-164.468, -64.902, -82.555, 18.247, 58.783, -9.697]
  Call Extruder(4796.57249)
  MoveL 397 to (41.5, -9.47, 25) mm, rotated rx 180 ry 0 rz 180 deg; joints [-163.355, -65.204, -81.56, 19.669, 58.323, -10.631]
  Call Extruder(4811.46836)
  MoveL 398 to (42.57, 0, 25) mm, rotated rx 180 ry 0 rz 180 deg; joints [-162.12, -65.419, -80.862, 21.199, 58.11, -11.58]
  Call Extruder(4826.36423)
  MoveL 399 to (41.5, 9.47, 25) mm, rotated rx 180 ry 0 rz 180 deg; joints [-160.81, -65.534, -80.497, 22.766, 58.149, -12.487]
  Call Extruder(4841.25990)
  MoveL 400 to (38.36, 18.47, 25) mm, rotated rx 180 ry 0 rz 180 deg; joints [-159.475, -65.539, -80.479, 24.299, 58.436, -13.297]
  Call Extruder(4856.15574)
  MoveL 401 to (33.29, 26.54, 25) mm, rotated rx -180 ry 0 rz 180 deg; joints [-158.16, -65.435, -80.811, 25.735, 58.953, -13.961]
  Call Extruder(4871.05156)
  MoveL 402 to (26.54, 33.28, 25) mm, rotated rx 180 ry 0 rz 180 deg; joints [-156.916, -65.23, -81.476, 27.017, 59.67, -14.44]
  Call Extruder(4885.94741)
  MoveL 403 to (18.47, 38.36, 25) mm, rotated rx -180 ry 0 rz -180 deg; joints [-155.789, -64.935, -82.444, 28.096, 60.55, -14.707]
  Call Extruder(4900.84307)
  MoveL 404 to (9.47, 41.51, 25) mm, rotated rx 180 ry 0 rz 180 deg; joints [-154.828, -64.571, -83.67, 28.931, 61.551, -14.751]
  Call Extruder(4915.73894)
  MoveL 405 to (0, 42.57, 25) mm, rotated rx 180 ry 0 rz -180 deg; joints [-154.081, -64.16, -85.094, 29.486, 62.626, -14.574]
  Call Extruder(4930.63482)
  MoveL 406 to (-9.47, 41.51, 25) mm, rotated rx -180 ry 0 rz 180 deg; joints [-153.594, -63.729, -86.652, 29.734, 63.725, -14.19]
  Call Extruder(4945.53047)
  MoveL 407 to (-18.47, 38.36, 25) mm, rotated rx -180 ry 0 rz 180 deg; joints [-153.408, -63.3, -88.267, 29.65, 64.801, -13.624]
  Call Extruder(4960.42632)
  MoveL 408 to (-26.54, 33.28, 25) mm, rotated rx -180 ry 0 rz -180 deg; joints [-153.557, -62.899, -89.861, 29.221, 65.806, -12.912]
  Call Extruder(4975.32214)
  MoveL 409 to (-33.28, 26.54, 25) mm, rotated rx 180 ry 0 rz 180 deg; joints [-154.059, -62.544, -91.354, 28.445, 66.694, -12.097]
  Call Extruder(4990.21799)
  MoveL 410 to (-38.36, 18.47, 25) mm, rotated rx -180 ry 0 rz 180 deg; joints [-154.913, -62.248, -92.667, 27.335, 67.421, -11.226]
  Call Extruder(5005.11365)
  MoveL 411 to (-41.5, 9.47, 25) mm, rotated rx 180 ry 0 rz 180 deg; joints [-156.091, -62.022, -93.73, 25.93, 67.949, -10.345]
  Call Extruder(5020.00952)
  MoveL 412 to (-42.57, 0, 25) mm, rotated rx -180 ry 0 rz -180 deg; joints [-157.533, -61.869, -94.483, 24.297, 68.243, -9.5]
  Call Extruder(5027.56380)
  MoveL 413 to (-42.03, -4.8, 25) mm, rotated rx 180 ry 0 rz 180 deg; joints [-158.35, -61.828, -94.689, 23.401, 68.263, -9.106]
  Set speed (130.0 mm/s)
  MoveL 414 to (-54.1, -7.67, 25) mm, rotated rx 180 ry 0 rz -180 deg; joints [-158.024, -61.47, -96.618, 23.507, 69.753, -8.56]
  Call Extruder(5031.63643)
  Set speed (30.0 mm/s)
  MoveL 415 to (-53.59, -12.23, 25) mm, rotated rx 180 ry 0 rz 180 deg; joints [-158.835, -61.438, -96.804, 22.63, 69.777, -8.2]
  Call Extruder(5042.56656)
  MoveL 416 to (-49.52, -23.85, 25) mm, rotated rx -180 ry 0 rz 180 deg; joints [-161.095, -61.434, -96.829, 20.238, 69.49, -7.361]
  Call Extruder(5053.49684)
  MoveL 417 to (-42.98, -34.27, 25) mm, rotated rx 180 ry 0 rz -180 deg; joints [-163.275, -61.517, -96.355, 17.972, 68.854, -6.675]
  Call Extruder(5064.42696)
  MoveL 418 to (-34.27, -42.98, 25) mm, rotated rx -180 ry 0 rz 180 deg; joints [-165.21, -61.689, -95.412, 15.993, 67.901, -6.154]
  Call Extruder(5075.35725)
  MoveL 419 to (-23.85, -49.53, 25) mm, rotated rx 180 ry 0 rz 180 deg; joints [-166.774, -61.955, -94.06, 14.426, 66.689, -5.813]
  Call Extruder(5086.28738)
  MoveL 420 to (-12.23, -53.59, 25) mm, rotated rx 180 ry 0 rz 180 deg; joints [-167.889, -62.312, -92.377, 13.353, 65.291, -5.667]
  Call Extruder(5097.21760)
  MoveL 421 to (0, -54.97, 25) mm, rotated rx -180 ry 0 rz 180 deg; joints [-168.526, -62.754, -90.459, 12.81, 63.79, -5.735]
  Call Extruder(5098.39508)
  MoveL 422 to (1.32, -54.82, 25) mm, rotated rx 180 ry 0 rz 180 deg; joints [-168.545, -62.807, -90.24, 12.807, 63.626, -5.766]
  Call Extruder(5108.14782)
  MoveL 423 to (12.23, -53.59, 25) mm, rotated rx 180 ry 0 rz 180 deg; joints [-168.697, -63.265, -88.406, 12.793, 62.268, -6.032]
  Call Extruder(5119.07797)
  MoveL 424 to (23.85, -49.53, 25) mm, rotated rx -180 ry 0 rz 180 deg; joints [-168.436, -63.819, -86.322, 13.275, 60.806, -6.565]
  Call Extruder(5130.00824)
  MoveL 425 to (34.27, -42.98, 25) mm, rotated rx 180 ry 0 rz 180 deg; joints [-167.797, -64.386, -84.306, 14.204, 59.476, -7.326]
  Call Extruder(5140.93837)
  MoveL 426 to (42.98, -34.27, 25) mm, rotated rx 180 ry 0 rz 180 deg; joints [-166.837, -64.932, -82.455, 15.517, 58.345, -8.29]
  Call Extruder(5151.86865)
  MoveL 427 to (49.52, -23.85, 25) mm, rotated rx -180 ry 0 rz 180 deg; joints [-165.618, -65.422, -80.853, 17.134, 57.466, -9.414]
  Call Extruder(5162.79878)
  MoveL 428 to (53.59, -12.23, 25) mm, rotated rx 180 ry 0 rz -180 deg; joints [-164.2, -65.825, -79.575, 18.971, 56.88, -10.638]
  Call Extruder(5173.72900)
  MoveL 429 to (54.97, 0, 25) mm, rotated rx 180 ry 0 rz 180 deg; joints [-162.641, -66.113, -78.68, 20.936, 56.614, -11.889]
  Call Extruder(5184.65923)
  MoveL 430 to (53.59, 12.23, 25) mm, rotated rx -180 ry 0 rz 180 deg; joints [-160.996, -66.265, -78.211, 22.936, 56.676, -13.087]
  Call Extruder(5195.58937)
  MoveL 431 to (49.52, 23.85, 25) mm, rotated rx -180 ry 0 rz -180 deg; joints [-159.322, -66.273, -78.188, 24.883, 57.056, -14.157]
  Call Extruder(5206.51964)
  MoveL 432 to (42.98, 34.27, 25) mm, rotated rx -180 ry 0 rz 180 deg; joints [-157.673, -66.134, -78.614, 26.698, 57.731, -15.03]
  Call Extruder(5217.44977)
  MoveL 433 to (34.27, 42.98, 25) mm, rotated rx -180 ry 0 rz 180 deg; joints [-156.102, -65.859, -79.468, 28.314, 58.66, -15.654]
  Call Extruder(5228.38004)
  MoveL 434 to (23.85, 49.52, 25) mm, rotated rx 180 ry 0 rz 180 deg; joints [-154.667, -65.467, -80.711, 29.676, 59.795, -15.997]
  Call Extruder(5239.31019)
  MoveL 435 to (12.23, 53.59, 25) mm, rotated rx 180 ry 0 rz 180 deg; joints [-153.426, -64.984, -82.283, 30.737, 61.079, -16.043]
  Call Extruder(5250.24041)
  MoveL 436 to (0, 54.97, 25) mm, rotated rx -180 ry 0 rz -180 deg; joints [-152.438, -64.441, -84.114, 31.458, 62.453, -15.798]
  Call Extruder(5261.17063)
  MoveL 437 to (-12.23, 53.59, 25) mm, rotated rx -180 ry 0 rz 180 deg; joints [-151.764, -63.875, -86.117, 31.804, 63.857, -15.282]
  Call Extruder(5272.10077)
  MoveL 438 to (-23.85, 49.52, 25) mm, rotated rx -180 ry 0 rz 180 deg; joints [-151.463, -63.318, -88.199, 31.744, 65.231, -14.531]
  Call Extruder(5283.03105)
  MoveL 439 to (-34.27, 42.98, 25) mm, rotated rx 180 ry 0 rz 180 deg; joints [-151.589, -62.802, -90.26, 31.249, 66.518, -13.592]
  Call Extruder(5293.96117)
  MoveL 440 to (-42.98, 34.27, 25) mm, rotated rx 180 ry 0 rz -180 deg; joints [-152.179, -62.352, -92.196, 30.303, 67.662, -12.523]
  Call Extruder(5304.89145)
  MoveL 441 to (-49.52, 23.85, 25) mm, rotated rx 180 ry 0 rz 180 deg; joints [-153.248, -61.986, -93.906, 28.91, 68.609, -11.389]
  Call Extruder(5315.82159)
  MoveL 442 to (-53.59, 12.23, 25) mm, rotated rx 180 ry 0 rz 180 deg; joints [-154.769, -61.711, -95.295, 27.107, 69.307, -10.253]
  Call Extruder(5326.75181)
  MoveL 443 to (-54.97, 0, 25) mm, rotated rx -180 ry 0 rz -180 deg; joints [-156.673, -61.53, -96.281, 24.973, 69.709, -9.175]
  Call Extruder(5332.27743)
  MoveL 444 to (-54.27, -6.18, 25) mm, rotated rx 180 ry 0 rz 180 deg; joints [-157.76, -61.481, -96.555, 23.793, 69.745, -8.679]
  Set speed (130.0 mm/s)
  MoveL 445 to (-49.9, -9.51, 25) mm, rotated rx 180 ry 0 rz 180 deg; joints [-158.616, -61.56, -96.114, 22.943, 69.285, -8.516]
  MoveL 446 to (2.97, -12.99, 25) mm, rotated rx 180 ry 0 rz -180 deg; joints [-162.152, -63.319, -88.194, 20.12, 63, -9.443]
  Call Extruder(5336.94099)
  Set speed (80.0 mm/s)
  MoveL 447 to (5.78, -12.01, 25) mm, rotated rx 180 ry 0 rz 180 deg; joints [-162.141, -63.452, -87.687, 20.199, 62.65, -9.594]
  Call Extruder(5341.60461)
  MoveL 448 to (8.31, -10.42, 25) mm, rotated rx -180 ry 0 rz -180 deg; joints [-162.027, -63.583, -87.193, 20.391, 62.328, -9.794]
  Call Extruder(5346.26881)
  MoveL 449 to (10.42, -8.31, 25) mm, rotated rx -180 ry 0 rz 180 deg; joints [-161.819, -63.706, -86.736, 20.684, 62.051, -10.035]
  Call Extruder(5350.93244)
  MoveL 450 to (12.01, -5.78, 25) mm, rotated rx 180 ry 0 rz 180 deg; joints [-161.529, -63.814, -86.339, 21.063, 61.833, -10.304]
  Call Extruder(5355.59601)
  MoveL 451 to (12.99, -2.97, 25) mm, rotated rx 180 ry 0 rz -180 deg; joints [-161.171, -63.901, -86.022, 21.507, 61.683, -10.587]
  Call Extruder(5360.25995)
  MoveL 452 to (13.33, 0, 25) mm, rotated rx 180 ry 0 rz 180 deg; joints [-160.763, -63.963, -85.799, 21.995, 61.61, -10.872]
  Call Extruder(5364.92391)
  MoveL 453 to (12.99, 2.97, 25) mm, rotated rx 180 ry 0 rz 180 deg; joints [-160.324, -63.995, -85.682, 22.502, 61.615, -11.141]
  Call Extruder(5369.58749)
  MoveL 454 to (12.01, 5.78, 25) mm, rotated rx 180 ry 0 rz -180 deg; joints [-159.874, -63.997, -85.677, 23.004, 61.7, -11.381]
  Call Extruder(5374.25111)
  MoveL 455 to (10.42, 8.31, 25) mm, rotated rx 180 ry 0 rz 180 deg; joints [-159.432, -63.967, -85.783, 23.479, 61.858, -11.578]
  Call Extruder(5378.91530)
  MoveL 456 to (8.31, 10.42, 25) mm, rotated rx 180 ry 0 rz 180 deg; joints [-159.021, -63.908, -85.995, 23.903, 62.082, -11.723]
  Call Extruder(5383.57892)
  MoveL 457 to (5.78, 12.01, 25) mm, rotated rx 180 ry 0 rz 180 deg; joints [-158.657, -63.823, -86.304, 24.257, 62.36, -11.808]
  Call Extruder(5388.24250)
  MoveL 458 to (2.97, 12.99, 25) mm, rotated rx 180 ry 0 rz 180 deg; joints [-158.359, -63.717, -86.694, 24.525, 62.679, -11.827]
  Call Extruder(5392.90645)
  MoveL 459 to (0, 13.33, 25) mm, rotated rx -180 ry 0 rz -180 deg; joints [-158.143, -63.595, -87.146, 24.693, 63.024, -11.781]
  Call Extruder(5397.57040)
  MoveL 460 to (-2.97, 13, 25) mm, rotated rx 180 ry 0 rz 180 deg; joints [-158.019, -63.465, -87.637, 24.752, 63.377, -11.673]
  Call Extruder(5402.23397)
  MoveL 461 to (-5.78, 12.01, 25) mm, rotated rx -180 ry 0 rz -180 deg; joints [-157.997, -63.332, -88.144, 24.698, 63.721, -11.509]
  Call Extruder(5406.89760)
  MoveL 462 to (-8.31, 10.42, 25) mm, rotated rx -180 ry 0 rz 180 deg; joints [-158.08, -63.204, -88.641, 24.532, 64.04, -11.298]
  Call Extruder(5411.56179)
  MoveL 463 to (-10.42, 8.31, 25) mm, rotated rx 180 ry 0 rz 180 deg; joints [-158.266, -63.087, -89.103, 24.26, 64.318, -11.051]
  Call Extruder(5416.22542)
  MoveL 464 to (-12.01, 5.78, 25) mm, rotated rx 180 ry 0 rz 180 deg; joints [-158.549, -62.986, -89.506, 23.894, 64.541, -10.782]
  Call Extruder(5420.88899)
  MoveL 465 to (-13, 2.97, 25) mm, rotated rx 180 ry 0 rz -180 deg; joints [-158.913, -62.907, -89.831, 23.451, 64.697, -10.504]
  Call Extruder(5425.55294)
  MoveL 466 to (-13.33, 0, 25) mm, rotated rx 180 ry 0 rz 180 deg; joints [-159.341, -62.851, -90.059, 22.953, 64.779, -10.23]
  Call Extruder(5430.21690)
  MoveL 467 to (-12.99, -2.97, 25) mm, rotated rx 180 ry 0 rz 180 deg; joints [-159.811, -62.822, -90.179, 22.426, 64.78, -9.973]
  Call Extruder(5434.88046)
  MoveL 468 to (-12.01, -5.78, 25) mm, rotated rx 180 ry 0 rz 180 deg; joints [-160.294, -62.82, -90.184, 21.898, 64.701, -9.747]
  Call Extruder(5439.54409)
  MoveL 469 to (-10.42, -8.31, 25) mm, rotated rx 180 ry 0 rz -180 deg; joints [-160.766, -62.847, -90.075, 21.398, 64.546, -9.56]
  Call Extruder(5444.20828)
  MoveL 470 to (-8.31, -10.42, 25) mm, rotated rx 180 ry 0 rz 180 deg; joints [-161.2, -62.9, -89.858, 20.952, 64.321, -9.421]
  Call Extruder(5448.87191)
  MoveL 471 to (-5.78, -12.01, 25) mm, rotated rx -180 ry 0 rz 180 deg; joints [-161.572, -62.978, -89.542, 20.585, 64.038, -9.337]
  Call Extruder(5453.53548)
  MoveL 472 to (-2.97, -13, 25) mm, rotated rx 180 ry 0 rz 180 deg; joints [-161.863, -63.076, -89.146, 20.317, 63.712, -9.312]
  Call Extruder(5458.19943)
  MoveL 473 to (0, -13.33, 25) mm, rotated rx -180 ry 0 rz -180 deg; joints [-162.059, -63.192, -88.689, 20.159, 63.36, -9.348]
  Call Extruder(5462.86339)
  MoveL 474 to (2.97, -12.99, 25) mm, rotated rx 180 ry 0 rz -180 deg; joints [-162.152, -63.319, -88.194, 20.12, 63, -9.443]
  Set speed (130.0 mm/s)
  MoveL 475 to (2.97, -12.99, 30) mm, rotated rx 180 ry 0 rz -180 deg; joints [-162.152, -62.551, -88.642, 20.176, 62.699, -9.567]
  MoveL 476 to (-26.25, -4.54, 30) mm, rotated rx 180 ry 0 rz 180 deg; joints [-159.288, -61.535, -92.766, 22.763, 66.07, -9.659]
  Call Extruder(5465.09602)
  Set speed (60.0 mm/s)
  MoveL 477 to (-26.09, -5.96, 30) mm, rotated rx -180 ry 0 rz 180 deg; joints [-159.522, -61.522, -92.823, 22.504, 66.072, -9.538]
  Call Extruder(5474.46081)
  MoveL 478 to (-24.12, -11.61, 30) mm, rotated rx 180 ry 0 rz -180 deg; joints [-160.532, -61.519, -92.835, 21.412, 65.917, -9.091]
  Call Extruder(5483.82573)
  MoveL 479 to (-20.93, -16.69, 30) mm, rotated rx 180 ry 0 rz 180 deg; joints [-161.513, -61.57, -92.612, 20.376, 65.604, -8.722]
  Call Extruder(5493.19094)
  MoveL 480 to (-16.69, -20.93, 30) mm, rotated rx -180 ry 0 rz 180 deg; joints [-162.406, -61.673, -92.168, 19.458, 65.15, -8.445]
  Call Extruder(5502.55586)
  MoveL 481 to (-11.61, -24.12, 30) mm, rotated rx -180 ry 0 rz 180 deg; joints [-163.159, -61.824, -91.526, 18.71, 64.577, -8.272]
  Call Extruder(5511.92064)
  MoveL 482 to (-5.96, -26.09, 30) mm, rotated rx -180 ry 0 rz -180 deg; joints [-163.733, -62.02, -90.721, 18.172, 63.917, -8.212]
  Call Extruder(5521.28575)
  MoveL 483 to (0, -26.77, 30) mm, rotated rx -180 ry 0 rz 180 deg; joints [-164.103, -62.252, -89.796, 17.87, 63.205, -8.27]
  Call Extruder(5530.65085)
  MoveL 484 to (5.96, -26.09, 30) mm, rotated rx 180 ry 0 rz 180 deg; joints [-164.258, -62.51, -88.799, 17.814, 62.478, -8.446]
  Call Extruder(5540.01565)
  MoveL 485 to (11.61, -24.11, 30) mm, rotated rx 180 ry 0 rz 180 deg; joints [-164.201, -62.782, -87.78, 17.999, 61.776, -8.735]
  Call Extruder(5549.38057)
  MoveL 486 to (16.69, -20.93, 30) mm, rotated rx 180 ry 0 rz 180 deg; joints [-163.944, -63.054, -86.789, 18.41, 61.134, -9.129]
  Call Extruder(5558.74577)
  MoveL 487 to (20.93, -16.69, 30) mm, rotated rx 180 ry 0 rz 180 deg; joints [-163.508, -63.312, -85.876, 19.02, 60.584, -9.61]
  Call Extruder(5568.11069)
  MoveL 488 to (24.12, -11.61, 30) mm, rotated rx 180 ry 0 rz 180 deg; joints [-162.92, -63.54, -85.085, 19.793, 60.153, -10.155]
  Call Extruder(5577.47549)
  MoveL 489 to (26.09, -5.96, 30) mm, rotated rx 180 ry 0 rz -180 deg; joints [-162.209, -63.725, -84.452, 20.689, 59.862, -10.736]
  Call Extruder(5586.84059)
  MoveL 490 to (26.77, 0, 30) mm, rotated rx 180 ry 0 rz -180 deg; joints [-161.41, -63.856, -84.009, 21.662, 59.725, -11.323]
  Call Extruder(5596.20569)
  MoveL 491 to (26.09, 5.96, 30) mm, rotated rx 180 ry 0 rz 180 deg; joints [-160.556, -63.926, -83.777, 22.667, 59.746, -11.883]
  Call Extruder(5605.57050)
  MoveL 492 to (24.12, 11.61, 30) mm, rotated rx 180 ry 0 rz 180 deg; joints [-159.683, -63.929, -83.766, 23.656, 59.922, -12.382]
  Call Extruder(5614.93541)
  MoveL 493 to (20.93, 16.69, 30) mm, rotated rx 180 ry 0 rz 180 deg; joints [-158.826, -63.866, -83.977, 24.587, 60.244, -12.794]
  Call Extruder(5624.30062)
  MoveL 494 to (16.69, 20.93, 30) mm, rotated rx -180 ry 0 rz 180 deg; joints [-158.019, -63.741, -84.399, 25.418, 60.694, -13.095]
  Call Extruder(5633.66553)
  MoveL 495 to (11.61, 24.11, 30) mm, rotated rx 180 ry 0 rz 180 deg; joints [-157.299, -63.56, -85.014, 26.116, 61.249, -13.268]
  Call Extruder(5643.03033)
  MoveL 496 to (5.96, 26.09, 30) mm, rotated rx 180 ry 0 rz 180 deg; joints [-156.697, -63.336, -85.792, 26.649, 61.883, -13.306]
  Call Extruder(5652.39544)
  MoveL 497 to (0, 26.77, 30) mm, rotated rx -180 ry 0 rz -180 deg; joints [-156.245, -63.081, -86.694, 26.993, 62.565, -13.208]
  Call Extruder(5661.76054)
  MoveL 498 to (-5.96, 26.09, 30) mm, rotated rx -180 ry 0 rz 180 deg; joints [-155.969, -62.809, -87.679, 27.128, 63.263, -12.98]
  Call Extruder(5671.12533)
  MoveL 499 to (-11.61, 24.12, 30) mm, rotated rx 180 ry 0 rz 180 deg; joints [-155.891, -62.537, -88.698, 27.045, 63.944, -12.639]
  Call Extruder(5680.49025)
  MoveL 500 to (-16.69, 20.93, 30) mm, rotated rx -180 ry 0 rz -180 deg; joints [-156.025, -62.276, -89.7, 26.738, 64.577, -12.204]
  Call Extruder(5689.85546)
  MoveL 501 to (-20.93, 16.69, 30) mm, rotated rx 180 ry 0 rz 180 deg; joints [-156.374, -62.042, -90.634, 26.215, 65.131, -11.699]
  Call Extruder(5699.22037)
  MoveL 502 to (-24.11, 11.61, 30) mm, rotated rx 180 ry 0 rz 180 deg; joints [-156.928, -61.842, -91.453, 25.493, 65.578, -11.152]
  Call Extruder(5708.58517)
  MoveL 503 to (-26.09, 5.96, 30) mm, rotated rx 180 ry 0 rz 180 deg; joints [-157.665, -61.686, -92.113, 24.603, 65.895, -10.592]
  Call Extruder(5717.95028)
  MoveL 504 to (-26.77, 0, 30) mm, rotated rx 180 ry 0 rz 180 deg; joints [-158.546, -61.578, -92.578, 23.589, 66.064, -10.046]
  Call Extruder(5722.73901)
  MoveL 505 to (-26.42, -3.05, 30) mm, rotated rx 180 ry 0 rz -180 deg; joints [-159.044, -61.549, -92.705, 23.035, 66.068, -9.786]
  Set speed (130.0 mm/s)
  MoveL 506 to (-41.86, -6.3, 30) mm, rotated rx 180 ry 0 rz 180 deg; joints [-158.606, -61.009, -95.213, 23.177, 67.95, -9.131]
  Call Extruder(5727.73686)
  Set speed (60.0 mm/s)
  MoveL 507 to (-41.5, -9.47, 30) mm, rotated rx 180 ry 0 rz 180 deg; joints [-159.151, -60.983, -95.341, 22.579, 67.959, -8.87]
  Call Extruder(5742.63251)
  MoveL 508 to (-38.36, -18.47, 30) mm, rotated rx 180 ry 0 rz 180 deg; joints [-160.835, -60.979, -95.361, 20.779, 67.723, -8.185]
  Call Extruder(5757.52836)
  MoveL 509 to (-33.28, -26.54, 30) mm, rotated rx 180 ry 0 rz 180 deg; joints [-162.466, -61.052, -94.999, 19.071, 67.228, -7.622]
  Call Extruder(5772.42418)
  MoveL 510 to (-26.54, -33.28, 30) mm, rotated rx 180 ry 0 rz -180 deg; joints [-163.93, -61.202, -94.279, 17.569, 66.498, -7.196]
  Call Extruder(5787.32003)
  MoveL 511 to (-18.47, -38.36, 30) mm, rotated rx 180 ry 0 rz 180 deg; joints [-165.137, -61.428, -93.242, 16.363, 65.574, -6.923]
  Call Extruder(5802.21568)
  MoveL 512 to (-9.47, -41.51, 30) mm, rotated rx -180 ry 0 rz 180 deg; joints [-166.024, -61.725, -91.947, 15.519, 64.508, -6.815]
  Call Extruder(5817.11155)
  MoveL 513 to (0, -42.57, 30) mm, rotated rx -180 ry 0 rz -180 deg; joints [-166.562, -62.083, -90.466, 15.07, 63.361, -6.884]
  Call Extruder(5832.00743)
  MoveL 514 to (9.47, -41.51, 30) mm, rotated rx 180 ry 0 rz 180 deg; joints [-166.745, -62.49, -88.876, 15.023, 62.196, -7.136]
  Call Extruder(5846.90309)
  MoveL 515 to (18.47, -38.36, 30) mm, rotated rx -180 ry 0 rz 180 deg; joints [-166.591, -62.925, -87.257, 15.364, 61.073, -7.571]
  Call Extruder(5861.79893)
  MoveL 516 to (26.54, -33.28, 30) mm, rotated rx 180 ry 0 rz -180 deg; joints [-166.133, -63.365, -85.688, 16.058, 60.05, -8.178]
  Call Extruder(5876.69475)
  MoveL 517 to (33.28, -26.54, 30) mm, rotated rx 180 ry 0 rz 180 deg; joints [-165.409, -63.786, -84.246, 17.058, 59.178, -8.935]
  Call Extruder(5891.59061)
  MoveL 518 to (38.36, -18.47, 30) mm, rotated rx 180 ry 0 rz 180 deg; joints [-164.468, -64.162, -82.997, 18.304, 58.499, -9.807]
  Call Extruder(5906.48626)
  MoveL 519 to (41.5, -9.47, 30) mm, rotated rx 180 ry 0 rz 180 deg; joints [-163.355, -64.468, -82.001, 19.731, 58.046, -10.748]
  Call Extruder(5921.38213)
  MoveL 520 to (42.57, 0, 30) mm, rotated rx 180 ry 0 rz 180 deg; joints [-162.12, -64.687, -81.303, 21.265, 57.838, -11.704]
  Call Extruder(5936.27800)
  MoveL 521 to (41.51, 9.47, 30) mm, rotated rx 180 ry 0 rz 180 deg; joints [-160.81, -64.803, -80.937, 22.836, 57.882, -12.62]
  Call Extruder(5951.17367)
  MoveL 522 to (38.36, 18.47, 30) mm, rotated rx 180 ry 0 rz 180 deg; joints [-159.475, -64.808, -80.92, 24.373, 58.172, -13.438]
  Call Extruder(5966.06951)
  MoveL 523 to (33.29, 26.54, 30) mm, rotated rx 180 ry 0 rz 180 deg; joints [-158.16, -64.703, -81.252, 25.812, 58.69, -14.109]
  Call Extruder(5980.96533)
  MoveL 524 to (26.54, 33.28, 30) mm, rotated rx 180 ry 0 rz 180 deg; joints [-156.916, -64.494, -81.917, 27.096, 59.408, -14.595]
  Call Extruder(5995.86118)
  MoveL 525 to (18.47, 38.36, 30) mm, rotated rx -180 ry 0 rz -180 deg; joints [-155.789, -64.195, -82.886, 28.176, 60.288, -14.869]
  Call Extruder(6010.75684)
  MoveL 526 to (9.47, 41.51, 30) mm, rotated rx 180 ry 0 rz 180 deg; joints [-154.828, -63.826, -84.112, 29.011, 61.287, -14.918]
  Call Extruder(6025.65271)
  MoveL 527 to (0, 42.57, 30) mm, rotated rx -180 ry 0 rz 180 deg; joints [-154.081, -63.408, -85.538, 29.565, 62.358, -14.745]
  Call Extruder(6040.54859)
  MoveL 528 to (-9.47, 41.51, 30) mm, rotated rx -180 ry 0 rz 180 deg; joints [-153.594, -62.969, -87.097, 29.811, 63.453, -14.364]
  Call Extruder(6055.44424)
  MoveL 529 to (-18.47, 38.36, 30) mm, rotated rx -180 ry 0 rz 180 deg; joints [-153.408, -62.532, -88.715, 29.726, 64.523, -13.799]
  Call Extruder(6070.34009)
  MoveL 530 to (-26.54, 33.28, 30) mm, rotated rx -180 ry 0 rz -180 deg; joints [-153.557, -62.122, -90.312, 29.294, 65.521, -13.087]
  Call Extruder(6085.23591)
  MoveL 531 to (-33.28, 26.54, 30) mm, rotated rx 180 ry 0 rz 180 deg; joints [-154.059, -61.758, -91.807, 28.513, 66.401, -12.27]
  Call Extruder(6100.13175)
  MoveL 532 to (-38.36, 18.47, 30) mm, rotated rx 180 ry 0 rz 180 deg; joints [-154.913, -61.454, -93.124, 27.4, 67.121, -11.394]
  Call Extruder(6115.02742)
  MoveL 533 to (-41.51, 9.47, 30) mm, rotated rx 180 ry 0 rz 180 deg; joints [-156.091, -61.221, -94.189, 25.992, 67.641, -10.507]
  Call Extruder(6129.92329)
  MoveL 534 to (-42.57, 0, 30) mm, rotated rx 180 ry 0 rz -180 deg; joints [-157.533, -61.063, -94.943, 24.354, 67.928, -9.653]
  Call Extruder(6137.47756)
  MoveL 535 to (-42.03, -4.8, 30) mm, rotated rx -180 ry 0 rz 180 deg; joints [-158.35, -61.021, -95.151, 23.457, 67.945, -9.254]
  Set speed (130.0 mm/s)
  MoveL 536 to (-54.1, -7.67, 30) mm, rotated rx 180 ry 0 rz 180 deg; joints [-158.024, -60.65, -97.084, 23.56, 69.428, -8.711]
  Call Extruder(6141.55020)
  Set speed (30.0 mm/s)
  MoveL 537 to (-53.59, -12.23, 30) mm, rotated rx -180 ry 0 rz -180 deg; joints [-158.835, -60.616, -97.271, 22.681, 69.449, -8.346]
  Call Extruder(6152.48033)
  MoveL 538 to (-49.53, -23.85, 30) mm, rotated rx 180 ry 0 rz 180 deg; joints [-161.095, -60.612, -97.296, 20.285, 69.157, -7.492]
  Call Extruder(6163.41061)
  MoveL 539 to (-42.98, -34.27, 30) mm, rotated rx 180 ry 0 rz 180 deg; joints [-163.275, -60.698, -96.82, 18.015, 68.518, -6.792]
  Call Extruder(6174.34073)
  MoveL 540 to (-34.27, -42.98, 30) mm, rotated rx 180 ry 0 rz 180 deg; joints [-165.21, -60.877, -95.875, 16.032, 67.565, -6.258]
  Call Extruder(6185.27102)
  MoveL 541 to (-23.85, -49.53, 30) mm, rotated rx 180 ry 0 rz -180 deg; joints [-166.774, -61.151, -94.519, 14.463, 66.356, -5.906]
  Call Extruder(6196.20115)
  MoveL 542 to (-12.23, -53.59, 30) mm, rotated rx 180 ry 0 rz 180 deg; joints [-167.889, -61.52, -92.833, 13.39, 64.963, -5.752]
  Call Extruder(6207.13137)
  MoveL 543 to (0, -54.97, 30) mm, rotated rx -180 ry 0 rz 180 deg; joints [-168.526, -61.973, -90.911, 12.846, 63.469, -5.816]
  Call Extruder(6208.68168)
  MoveL 544 to (1.74, -54.77, 30) mm, rotated rx 180 ry 0 rz 180 deg; joints [-168.551, -62.045, -90.622, 12.842, 63.254, -5.858]
  Call Extruder(6218.06159)
  MoveL 545 to (12.23, -53.59, 30) mm, rotated rx 180 ry 0 rz 180 deg; joints [-168.697, -62.495, -88.854, 12.831, 61.955, -6.112]
  Call Extruder(6228.99173)
  MoveL 546 to (23.85, -49.53, 30) mm, rotated rx 180 ry 0 rz 180 deg; joints [-168.436, -63.06, -86.767, 13.315, 60.501, -6.647]
  Call Extruder(6239.92201)
  MoveL 547 to (34.27, -42.98, 30) mm, rotated rx 180 ry 0 rz 180 deg; joints [-167.797, -63.638, -84.75, 14.249, 59.181, -7.413]
  Call Extruder(6250.85213)
  MoveL 548 to (42.98, -34.27, 30) mm, rotated rx 180 ry 0 rz 180 deg; joints [-166.837, -64.192, -82.897, 15.566, 58.058, -8.384]
  Call Extruder(6261.78242)
  MoveL 549 to (49.53, -23.85, 30) mm, rotated rx 180 ry 0 rz 180 deg; joints [-165.618, -64.69, -81.294, 17.19, 57.187, -9.516]
  Call Extruder(6272.71255)
  MoveL 550 to (53.59, -12.23, 30) mm, rotated rx -180 ry 0 rz -180 deg; joints [-164.2, -65.098, -80.015, 19.033, 56.609, -10.75]
  Call Extruder(6283.64277)
  MoveL 551 to (54.97, 0, 30) mm, rotated rx 180 ry 0 rz 180 deg; joints [-162.641, -65.389, -79.12, 21.004, 56.349, -12.011]
  Call Extruder(6294.57299)
  MoveL 552 to (53.59, 12.23, 30) mm, rotated rx 180 ry 0 rz 180 deg; joints [-160.996, -65.544, -78.65, 23.009, 56.416, -13.219]
  Call Extruder(6305.50314)
  MoveL 553 to (49.52, 23.85, 30) mm, rotated rx 180 ry 0 rz -180 deg; joints [-159.322, -65.551, -78.628, 24.961, 56.801, -14.299]
  Call Extruder(6316.43341)
  MoveL 554 to (42.98, 34.27, 30) mm, rotated rx 180 ry 0 rz 180 deg; joints [-157.673, -65.411, -79.054, 26.779, 57.478, -15.181]
  Call Extruder(6327.36354)
  MoveL 555 to (34.27, 42.98, 30) mm, rotated rx 180 ry 0 rz 180 deg; joints [-156.102, -65.132, -79.908, 28.398, 58.408, -15.814]
  Call Extruder(6338.29381)
  MoveL 556 to (23.85, 49.52, 30) mm, rotated rx -180 ry 0 rz -180 deg; joints [-154.667, -64.735, -81.151, 29.76, 59.542, -16.164]
  Call Extruder(6349.22396)
  MoveL 557 to (12.23, 53.59, 30) mm, rotated rx 180 ry 0 rz 180 deg; joints [-153.426, -64.245, -82.725, 30.821, 60.824, -16.217]
  Call Extruder(6360.15418)
  MoveL 558 to (0, 54.97, 30) mm, rotated rx 180 ry 0 rz 180 deg; joints [-152.438, -63.694, -84.557, 31.541, 62.194, -15.978]
  Call Extruder(6371.08440)
  MoveL 559 to (-12.23, 53.59, 30) mm, rotated rx 180 ry 0 rz 180 deg; joints [-151.764, -63.118, -86.562, 31.886, 63.592, -15.466]
  Call Extruder(6382.01453)
  MoveL 560 to (-23.85, 49.52, 30) mm, rotated rx 180 ry 0 rz 180 deg; joints [-151.463, -62.55, -88.647, 31.822, 64.959, -14.717]
  Call Extruder(6392.94482)
  MoveL 561 to (-34.27, 42.98, 30) mm, rotated rx 180 ry 0 rz 180 deg; joints [-151.589, -62.023, -90.711, 31.323, 66.237, -13.778]
  Call Extruder(6403.87494)
  MoveL 562 to (-42.98, 34.27, 30) mm, rotated rx 180 ry 0 rz -180 deg; joints [-152.179, -61.561, -92.651, 30.373, 67.372, -12.707]
  Call Extruder(6414.80522)
  MoveL 563 to (-49.52, 23.85, 30) mm, rotated rx 180 ry 0 rz -180 deg; joints [-153.248, -61.184, -94.365, 28.976, 68.309, -11.567]
  Call Extruder(6425.73536)
  MoveL 564 to (-53.59, 12.23, 30) mm, rotated rx 180 ry 0 rz 180 deg; joints [-154.769, -60.9, -95.758, 27.168, 68.997, -10.423]
  Call Extruder(6436.66558)
  MoveL 565 to (-54.97, 0, 30) mm, rotated rx -180 ry 0 rz -180 deg; joints [-156.673, -60.712, -96.747, 25.028, 69.389, -9.334]
  Call Extruder(6442.19119)
  MoveL 566 to (-54.27, -6.18, 30) mm, rotated rx 180 ry 0 rz 180 deg; joints [-157.76, -60.661, -97.021, 23.846, 69.421, -8.831]
  Set speed (130.0 mm/s)
  MoveL 567 to (-49.9, -9.51, 30) mm, rotated rx -180 ry 0 rz 180 deg; joints [-158.616, -60.743, -96.579, 22.995, 68.96, -8.663]
  MoveL 568 to (2.97, -12.99, 30) mm, rotated rx 180 ry 0 rz -180 deg; joints [-162.152, -62.551, -88.642, 20.176, 62.699, -9.567]
  Call Extruder(6446.85477)
  Set speed (80.0 mm/s)
  MoveL 569 to (5.78, -12.01, 30) mm, rotated rx 180 ry 0 rz 180 deg; joints [-162.141, -62.686, -88.134, 20.256, 62.351, -9.718]
  Call Extruder(6451.51839)
  MoveL 570 to (8.31, -10.42, 30) mm, rotated rx 180 ry 0 rz -180 deg; joints [-162.027, -62.82, -87.639, 20.449, 62.032, -9.919]
  Call Extruder(6456.18258)
  MoveL 571 to (10.42, -8.31, 30) mm, rotated rx 180 ry 0 rz -180 deg; joints [-161.819, -62.945, -87.182, 20.743, 61.757, -10.161]
  Call Extruder(6460.84621)
  MoveL 572 to (12.01, -5.78, 30) mm, rotated rx 180 ry 0 rz 180 deg; joints [-161.529, -63.055, -86.785, 21.124, 61.541, -10.431]
  Call Extruder(6465.50978)
  MoveL 573 to (13, -2.97, 30) mm, rotated rx -180 ry 0 rz -180 deg; joints [-161.171, -63.144, -86.467, 21.569, 61.394, -10.718]
  Call Extruder(6470.17373)
  MoveL 574 to (13.33, 0, 30) mm, rotated rx -180 ry 0 rz 180 deg; joints [-160.763, -63.207, -86.244, 22.058, 61.322, -11.004]
  Call Extruder(6474.83769)
  MoveL 575 to (12.99, 2.97, 30) mm, rotated rx -180 ry 0 rz 180 deg; joints [-160.324, -63.24, -86.127, 22.567, 61.329, -11.276]
  Call Extruder(6479.50126)
  MoveL 576 to (12.01, 5.78, 30) mm, rotated rx 180 ry 0 rz -180 deg; joints [-159.874, -63.242, -86.122, 23.07, 61.414, -11.519]
  Call Extruder(6484.16488)
  MoveL 577 to (10.42, 8.31, 30) mm, rotated rx 180 ry 0 rz 180 deg; joints [-159.432, -63.212, -86.228, 23.546, 61.573, -11.719]
  Call Extruder(6488.82907)
  MoveL 578 to (8.31, 10.42, 30) mm, rotated rx -180 ry 0 rz 180 deg; joints [-159.021, -63.152, -86.44, 23.97, 61.797, -11.866]
  Call Extruder(6493.49269)
  MoveL 579 to (5.78, 12.01, 30) mm, rotated rx -180 ry 0 rz 180 deg; joints [-158.657, -63.065, -86.75, 24.325, 62.075, -11.953]
  Call Extruder(6498.15627)
  MoveL 580 to (2.97, 12.99, 30) mm, rotated rx 180 ry 0 rz 180 deg; joints [-158.359, -62.957, -87.14, 24.593, 62.393, -11.974]
  Call Extruder(6502.82023)
  MoveL 581 to (0, 13.33, 30) mm, rotated rx -180 ry 0 rz 180 deg; joints [-158.143, -62.833, -87.592, 24.76, 62.737, -11.93]
  Call Extruder(6507.48418)
  MoveL 582 to (-2.97, 12.99, 30) mm, rotated rx 180 ry 0 rz -180 deg; joints [-158.019, -62.7, -88.084, 24.819, 63.088, -11.823]
  Call Extruder(6512.14774)
  MoveL 583 to (-5.78, 12.01, 30) mm, rotated rx -180 ry 0 rz 180 deg; joints [-157.997, -62.565, -88.592, 24.765, 63.431, -11.659]
  Call Extruder(6516.81138)
  MoveL 584 to (-8.31, 10.42, 30) mm, rotated rx -180 ry 0 rz 180 deg; joints [-158.08, -62.434, -89.09, 24.598, 63.748, -11.447]
  Call Extruder(6521.47557)
  MoveL 585 to (-10.42, 8.31, 30) mm, rotated rx 180 ry 0 rz 180 deg; joints [-158.266, -62.314, -89.552, 24.325, 64.023, -11.199]
  Call Extruder(6526.13919)
  MoveL 586 to (-12.01, 5.78, 30) mm, rotated rx -180 ry 0 rz 180 deg; joints [-158.549, -62.211, -89.957, 23.957, 64.244, -10.928]
  Call Extruder(6530.80276)
  MoveL 587 to (-13, 2.97, 30) mm, rotated rx -180 ry 0 rz -180 deg; joints [-158.913, -62.129, -90.281, 23.513, 64.398, -10.648]
  Call Extruder(6535.46672)
  MoveL 588 to (-13.33, 0, 30) mm, rotated rx -180 ry 0 rz -180 deg; joints [-159.341, -62.072, -90.51, 23.014, 64.477, -10.371]
  Call Extruder(6540.13067)
  MoveL 589 to (-12.99, -2.97, 30) mm, rotated rx -180 ry 0 rz 180 deg; joints [-159.811, -62.043, -90.63, 22.485, 64.477, -10.112]
  Call Extruder(6544.79423)
  MoveL 590 to (-12.01, -5.78, 30) mm, rotated rx 180 ry 0 rz 180 deg; joints [-160.294, -62.041, -90.636, 21.956, 64.397, -9.882]
  Call Extruder(6549.45786)
  MoveL 591 to (-10.42, -8.31, 30) mm, rotated rx 180 ry 0 rz 180 deg; joints [-160.766, -62.068, -90.527, 21.455, 64.241, -9.692]
  Call Extruder(6554.12206)
  MoveL 592 to (-8.31, -10.42, 30) mm, rotated rx -180 ry 0 rz 180 deg; joints [-161.2, -62.123, -90.309, 21.009, 64.016, -9.551]
  Call Extruder(6558.78569)
  MoveL 593 to (-5.78, -12.01, 30) mm, rotated rx 180 ry 0 rz 180 deg; joints [-161.572, -62.202, -89.993, 20.642, 63.733, -9.465]
  Call Extruder(6563.44925)
  MoveL 594 to (-2.97, -13, 30) mm, rotated rx 180 ry 0 rz 180 deg; joints [-161.863, -62.303, -89.596, 20.373, 63.408, -9.438]
  Call Extruder(6568.11320)
  MoveL 595 to (0, -13.33, 30) mm, rotated rx -180 ry 0 rz -180 deg; joints [-162.059, -62.421, -89.138, 20.215, 63.058, -9.472]
  Call Extruder(6572.77716)
  MoveL 596 to (2.97, -12.99, 30) mm, rotated rx 180 ry 0 rz -180 deg; joints [-162.152, -62.551, -88.642, 20.176, 62.699, -9.567]
  Set speed (130.0 mm/s)
  MoveL 597 to (2.97, -12.99, 35) mm, rotated rx 180 ry 0 rz -180 deg; joints [-162.152, -61.783, -89.081, 20.235, 62.39, -9.695]
  MoveL 598 to (-26.25, -4.54, 35) mm, rotated rx -180 ry 0 rz 180 deg; joints [-159.288, -60.742, -93.213, 22.823, 65.751, -9.806]
  Call Extruder(6575.00979)
  Set speed (60.0 mm/s)
  MoveL 599 to (-26.09, -5.96, 35) mm, rotated rx 180 ry 0 rz 180 deg; joints [-159.522, -60.729, -93.27, 22.563, 65.752, -9.684]
  Call Extruder(6584.37457)
  MoveL 600 to (-24.11, -11.61, 35) mm, rotated rx -180 ry 0 rz 180 deg; joints [-160.532, -60.726, -93.282, 21.469, 65.595, -9.23]
  Call Extruder(6593.73950)
  MoveL 601 to (-20.93, -16.69, 35) mm, rotated rx 180 ry 0 rz 180 deg; joints [-161.513, -60.778, -93.059, 20.431, 65.281, -8.854]
  Call Extruder(6603.10470)
  MoveL 602 to (-16.69, -20.93, 35) mm, rotated rx 180 ry 0 rz -180 deg; joints [-162.406, -60.884, -92.613, 19.511, 64.826, -8.571]
  Call Extruder(6612.46962)
  MoveL 603 to (-11.61, -24.12, 35) mm, rotated rx 180 ry 0 rz 180 deg; joints [-163.159, -61.04, -91.97, 18.762, 64.254, -8.394]
  Call Extruder(6621.83441)
  MoveL 604 to (-5.96, -26.09, 35) mm, rotated rx 180 ry 0 rz 180 deg; joints [-163.733, -61.24, -91.164, 18.224, 63.596, -8.33]
  Call Extruder(6631.19953)
  MoveL 605 to (0, -26.77, 35) mm, rotated rx 180 ry 0 rz 180 deg; joints [-164.103, -61.477, -90.237, 17.922, 62.887, -8.385]
  Call Extruder(6640.56462)
  MoveL 606 to (5.96, -26.09, 35) mm, rotated rx 180 ry 0 rz 180 deg; joints [-164.258, -61.741, -89.238, 17.867, 62.165, -8.56]
  Call Extruder(6649.92942)
  MoveL 607 to (11.61, -24.11, 35) mm, rotated rx -180 ry 0 rz 180 deg; joints [-164.201, -62.019, -88.217, 18.054, 61.467, -8.85]
  Call Extruder(6659.29433)
  MoveL 608 to (16.69, -20.93, 35) mm, rotated rx 180 ry 0 rz 180 deg; joints [-163.944, -62.296, -87.226, 18.467, 60.829, -9.245]
  Call Extruder(6668.65954)
  MoveL 609 to (20.93, -16.69, 35) mm, rotated rx -180 ry 0 rz 180 deg; joints [-163.508, -62.559, -86.312, 19.079, 60.283, -9.729]
  Call Extruder(6678.02446)
  MoveL 610 to (24.12, -11.61, 35) mm, rotated rx 180 ry 0 rz 180 deg; joints [-162.92, -62.791, -85.519, 19.855, 59.857, -10.278]
  Call Extruder(6687.38926)
  MoveL 611 to (26.09, -5.96, 35) mm, rotated rx -180 ry 0 rz -180 deg; joints [-162.209, -62.979, -84.886, 20.754, 59.571, -10.864]
  Call Extruder(6696.75436)
  MoveL 612 to (26.77, 0, 35) mm, rotated rx -180 ry 0 rz -180 deg; joints [-161.41, -63.113, -84.443, 21.73, 59.436, -11.456]
  Call Extruder(6706.11946)
  MoveL 613 to (26.09, 5.96, 35) mm, rotated rx 180 ry 0 rz 180 deg; joints [-160.556, -63.183, -84.21, 22.737, 59.46, -12.021]
  Call Extruder(6715.48426)
  MoveL 614 to (24.12, 11.61, 35) mm, rotated rx 180 ry 0 rz 180 deg; joints [-159.683, -63.187, -84.199, 23.728, 59.639, -12.526]
  Call Extruder(6724.84918)
  MoveL 615 to (20.93, 16.69, 35) mm, rotated rx -180 ry 0 rz 180 deg; joints [-158.826, -63.123, -84.41, 24.661, 59.962, -12.943]
